// TIA Portal V20 export
// export: Created 2025-12-01T14:57:41.3483873Z, ExportSetting None, DisplayName Totally Integrated Automation Portal, DisplayVersion V20 Update 3, DisplayName TIA Portal Openness, DisplayVersion V20 Update 3, DisplayName TIA Portal Version Control Interface, DisplayVersion V20 Update 3, DisplayName STEP 7 Professional, DisplayVersion V20 Update 3, DisplayName STEP 7 Safety, DisplayVersion V20 Update 2, DisplayName WinCC Basic/Comfort/Advanced, DisplayVersion V20 Update 3, DisplayName WinCC Professional, DisplayVersion V20 Update 3, DisplayName WinCC Unified, DisplayVersion V20 Update 3
FUNCTION_BLOCK "FB380_PaletizadorLenze_NDD"   // FB380, LAD
{ S7_Optimized_Access := 'FALSE' }
// stored: AutoNumber false, SetENOAutomatically false
   VAR_INPUT
      MesaElevador : UInt;
      MesaHorquilla : UInt;
      MesaGarra : UInt;
      NDB_ConfigNDD : UInt;
      NDB_DatosNDD : UInt;
      NDB_Enfardadora : UInt;
      Error_Tx : Bool;
      DesHabilitar_MAQ : Bool;
      DesHabilitar_Enfadadora : Bool;
      DesHabilitar_Horquilla : Bool;   // DesHabilitar la Horquilla
      DesHabilitar_Garra : Bool;   // DesHabilitar la Garra
      PorCapas_Enfardado : Bool;
      Mantenimiento : Bool;
      TermicoFRENO_Elev : Bool;
      Elev_Protusion : Bool;
      EM_Elev_Down : Bool;
      CheckElev_EnEntrada : Bool;
      CheckElev_EnSalida : Bool;
      CheckElev_EnEnfardadora : Bool;
      CheckElev_EnHorquilla : Bool;
      CheckElev_EnGarra : Bool;
      EM_Elev_Up : Bool;
      EM_Elev_Bulon_Dch : Bool;
      EM_Elev_Bulon_Izq : Bool;
      P_Puesto_Capa : Bool;
      P_Puesto_Subir : Bool;
      P_Puesto_Bajar : Bool;
      BarreraNivelUp : Bool;
      BarreraNivelDown : Bool;
      Elev_Galibo_01 : Bool;
      Elev_Galibo_02 : Bool;
      Elev_Galibo_03 : Bool;
      Elev_Galibo_04 : Bool;
      Manual_ElevUp : Bool;
      Manual_ElevDown : Bool;
      Homming_Elev : Bool;
      ModoEncoder_Elev : Bool;
      pHsRef_Elev : Bool;
      V_TOut_Elevacion : Time;
      V_TMP_Protusion : Time;
   END_VAR
   VAR_OUTPUT
      DI3VarElev_pHsReferenciaCero : Bool;
      DesHabiBarreraNivelUP : Bool;
      DesHabiBarreraNivelDown : Bool;
   END_VAR
   VAR
      FB_Enfardadora { S7_SetPoint := 'True'} : "FB384_Enfardadora_Paletizador_NDD";
      Interlock_Horquilla { S7_SetPoint := 'True'} : "NDD_Interlock_Horquilla";
      Interlock_Garras { S7_SetPoint := 'True'} : "NDD_Interlock_Garras";
      Interlock_TELEV { S7_SetPoint := 'True'} : "NDD_Interlock_TElev";
      Ordenes { S7_SetPoint := 'True'} : "NDD_Ordenes";
      TMPEnPisoCarga { S7_SetPoint := 'True'} : TON_TIME;
      TMPEnPisoDesCarga { S7_SetPoint := 'True'} : TON_TIME;
      TMPEnPisoHorquilla { S7_SetPoint := 'True'} : TON_TIME;
      TMPEnPisoGarra { S7_SetPoint := 'True'} : TON_TIME;
      TMPEnPisoEnfradadora { S7_SetPoint := 'True'} : TON_TIME;
      TEstableMovElev { S7_SetPoint := 'True'} : TON_TIME;
      TMPGalibo { S7_SetPoint := 'True'} : TON_TIME;
      TMPProtusion { S7_SetPoint := 'True'} : TON_TIME;
      TOutElevacion { S7_SetPoint := 'True'} : TON_TIME;
      TEsperaMoverElev { S7_SetPoint := 'True'} : TON_TIME;
      TOutPosicion { S7_SetPoint := 'True'} : TON_TIME;
      VelocidadEnfardadora : Int;
      MemoAlturaPedido : Int;
      MemoEventoPaletizado : UInt;
      AlturaActualPedido : Int;
      PosicionCarga : Int;
      PosicionDesCarga : Int;
      PosicionEnfardado : Int;
      PosicionHorquilla : Int;
      PosicionGarra : Int;
      PosicionActual : Int;
      PosicionMoverElev : Int;
      PosicionUltimaElev : Int;
      ConsignaFR_elev : Int;
      SubjectArea_Elev : Word;
      IDArea_Elev : Word;
      MoverElev : Bool;
      FinMoverElev : Bool;
      MFinMoverElev : Bool;
      PosCarga_OK : Bool;
      PosDesCarga_OK : Bool;
      PosHorquilla_OK : Bool;
      PosGarra_OK : Bool;
      PosEnfardadora_OK : Bool;
      TestAuto_HorqGarra : Bool;
      ELEV_ET00 : Bool;
      ELEV_ET01 : Bool;
      CARGA_ET01 : Bool;
      CARGA_ET02 : Bool;
      CARGA_ET03 : Bool;
      CARGA_ET04 : Bool;
      CARGARRA_ET01 : Bool;
      CARGARRA_ET02 : Bool;
      CARGARRA_ET03 : Bool;
      CARGARRA_ET04 : Bool;
      CARGARRA_ET05 : Bool;
      DCARGARRA_ET01 : Bool;
      DCARGARRA_ET02 : Bool;
      DCARGARRA_ET03 : Bool;
      DCARGARRA_ET04 : Bool;
      DCARGARRA_ET05 : Bool;
      DCARHORQ_ET01 : Bool;
      DCARHORQ_ET02 : Bool;
      DCARHORQ_ET03 : Bool;
      DCARHORQ_ET04 : Bool;
      DCARHORQ_ET05 : Bool;
      PALETIZAR_ET01 : Bool;
      PALETIZAR_ET02 : Bool;
      PALETIZAR_ER01 : Bool;
      PALETIZAR_ER02 : Bool;
      DESCARGA_ET02 : Bool;
      DESCARGA_ET03 : Bool;
      DESCARGA_ET04 : Bool;
      DESCARGA_ET05 : Bool;
      DESCARGA_ET06 : Bool;
      MoverElev_Entrada : Bool;
      MoverElev_Garra : Bool;
      MoverElev_HorquillaUp : Bool;
      MoverElev_HorquillaDown : Bool;
      MoverElev_Enfardado : Bool;
      MoverElev_Salida : Bool;
      MoverElev_Puesto : Bool;
      HorqGarra_EnOperacion : Bool;
      Elev_EnReset : Bool;
      Elev_EnReposo : Bool;
      Elev_CargaDeEntrada : Bool;
      Elev_CargaDeGarra : Bool;
      Elev_DesCargaEnGarra : Bool;
      Elev_DesCargaEnHorquilla : Bool;
      Elev_DesCargaEnSalida : Bool;
      Elev_Paletizando : Bool;
      PuestoCarga_EnElev : Bool;
      Memo_NuevaCapa : Bool;
      MA_Puesto_NuevaCapa : Bool;
      MA_Puesto_Subir : Bool;
      MA_Puesto_Bajar : Bool;
      MA_Puesto_Baliza : Bool;
      LibreZonaAlta : Bool;
      ErrorVariador_Elev : Bool;
      MemoHoming_Elev : Bool;
      ReferenciaOK_Elev : Bool;
      MovHorq_Bloqueada : Bool;
      MovGarra_Bloqueada : Bool;
      ErrorControlPedido : Bool;
      AvisoControlPedido : Bool;
      EventoInicioPaletizado : Bool;
      EventoFinalPaletizado : Bool;
      EventoAlturaPedido : Bool;
      EventoInicioEnfardado : Bool;
      EventoFinalEnfardado : Bool;
      EventoErrorEnfradado : Bool;
   END_VAR
   VAR_TEMP
      EstadoZonaMaquina : "EstadoZona";
      EstadoZonaMesa : "EstadoZona";
      EstadoVI : "EstadosMesa_Transporte_Paletizador_NDD";
      EstadoMAQ : "EstadoMaquina_PaletizadorLenze_NDD";
      EstadoHorquilla : "EstadosMesa_HorquillaLenze_Paletizador_NDD";
      EstadoGarra : "EstadosMesa_GarrasLenze_Paletizador_NDD";
      DatosEscada : "UDT_ScadaDatosMaquina";
      EstadoZonaEnfa : "EstadoZona";
      EstadoZonaMovElev : "EstadoZona";
      NodoVar_Elev : "Status_NodosProfinet";
      P_EstadoZonaEnfa : DWord;
      P_EstadoZonaMovElev : DWord;
      P_NodoVar_Elev : DWord;
      Guardar_AR1 : DWord;
      Guardar_AR2 : DWord;
      P_Temporal : DWord;
      DB_ConfigNDD : Word;
      DB_DatosNDD : Word;
      NumDB_DiagProfinet : UInt;
      NumDB_DatosDanfoss : UInt;
      ByteInicial_VarElev : UInt;
      NumNodo_VarElev : UInt;
      VeloManual : Int;   // Velocidad Manual
      VeloCapa : Int;   // Velocidad Nueva Capa
      VeloRapidaDOWN : Int;   // Velocidad Rapida para ir a Posicion DOWN
      VeloLentaDOWN : Int;   // Velocidad Lenta para ir a Posicion DOWN
      PosLentaDOWN : Int;   // Diferencia para pasar Lenta para ir a Posicion DOWN
      VeloRapidaUP : Int;   // Velocidad Rapida para ir a Posicion UP
      VeloLentaUP : Int;   // Velocidad Lenta para ir a Posicion UP
      PosLentaUP : Int;   // Diferencia para pasar Lenta para ir a Posicion UP
      FactorVelocidadEnfardadora : Int;
      AltNivelCtr : Int;
      AlturaMax : Int;
      AlturaMin : Int;
      AlturaPaleta : Int;
      AlturaGalibo : Int;
      AlturaMaximoPedido : Int;
      AlturaControlPedido : Int;
      PosicionLibreNDD : Int;
      PosicionLibreHorq : Int;
      PosicionLibreGarra : Int;
      MemoPosActual_Elev : Int;
      MargenPos : Int;
      AuxPosMax : Int;
      AuxPosMin : Int;
      MargenPedido : Int;
      AuxAlturaPedidoMax : Int;
      AuxAlturaPedidoMin : Int;
      TempInt : Int;
      OrdenPosUP : Bool;
      OrdenPosDOWN : Bool;
      OrdenPosLentaUP : Bool;
      OrdenPosLentaDown : Bool;
      ZonaEnMarcha : Bool;
      ZonaEnReset : Bool;
      ZonaEnParoBlando : Bool;
      EnPisoAbajo : Bool;
      NodoNoPres_VarElev : Bool;
      AuxEstados : Bool;
      Etapas_OK : Bool;
      Transicion_OK : Bool;
      ControlPaleta_OK : Bool;
      AlturaMaxOK_Puesto : Bool;
      AlturaMinOK_Puesto : Bool;
      DesHabilitar_NDD : Bool;
      CalcularAlturaPedido : Bool;
   END_VAR
   VAR_TEMP   // added for the SCL form of the ladder/FBD networks
      _w1 : Bool;
      _w2 : Bool;
      _w3 : Bool;
      _w4 : Bool;
      _w5 : Bool;
      _w6 : Bool;
      _w7 : Bool;
   END_VAR
BEGIN

REGION Network 1: Variables de Testeo en Automatico
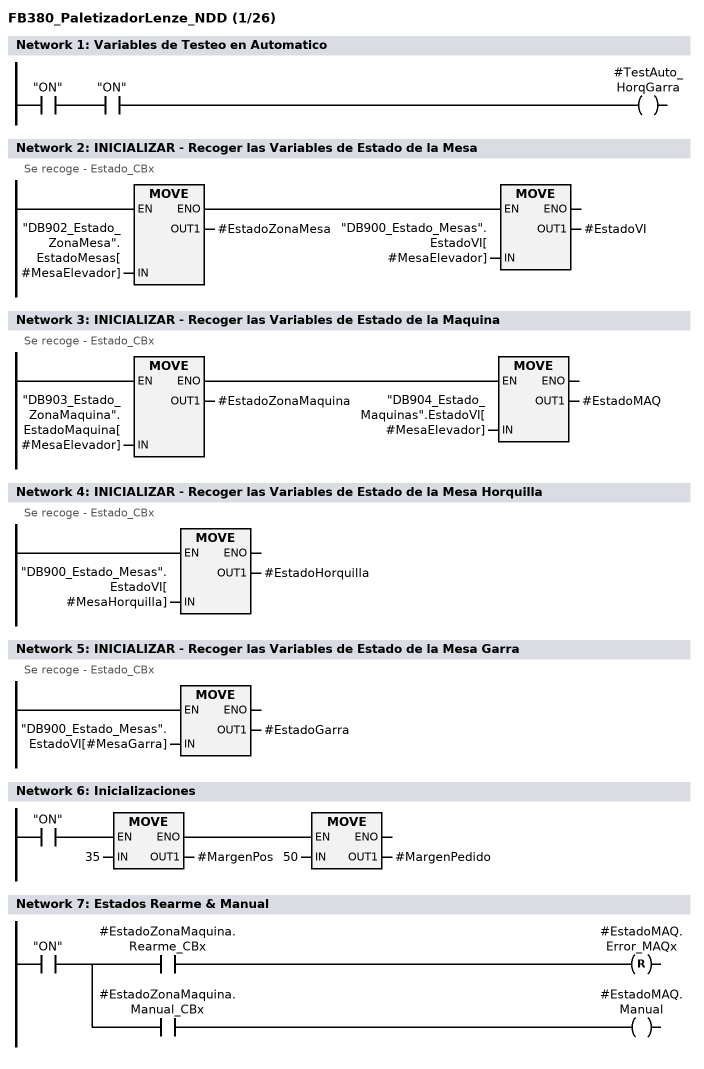
   RUNG wire#powerrail
      Contact( "ON" )
      Contact( "ON" )
      Coil( #TestAuto_HorqGarra )
   END_RUNG
   // the same network as SCL:
   #TestAuto_HorqGarra := "ON" AND "ON";
END_REGION

REGION Network 2: INICIALIZAR - Recoger las Variables de Estado de la Mesa
   // Se recoge - Estado_CBx
   RUNG wire#powerrail
      Move(in := "DB902_Estado_ZonaMesa".EstadoMesas[#MesaElevador], out1 => #EstadoZonaMesa)
      Move(in := "DB900_Estado_Mesas".EstadoVI[#MesaElevador], out1 => #EstadoVI)
   END_RUNG
   // the same network as SCL:
   #EstadoZonaMesa := "DB902_Estado_ZonaMesa".EstadoMesas[#MesaElevador];
   #EstadoVI := "DB900_Estado_Mesas".EstadoVI[#MesaElevador];
END_REGION

REGION Network 3: INICIALIZAR - Recoger las Variables de Estado de la Maquina
   // Se recoge - Estado_CBx
   RUNG wire#powerrail
      Move(in := "DB903_Estado_ZonaMaquina".EstadoMaquina[#MesaElevador], out1 => #EstadoZonaMaquina)
      Move(in := "DB904_Estado_Maquinas".EstadoVI[#MesaElevador], out1 => #EstadoMAQ)
   END_RUNG
   // the same network as SCL:
   #EstadoZonaMaquina := "DB903_Estado_ZonaMaquina".EstadoMaquina[#MesaElevador];
   #EstadoMAQ := "DB904_Estado_Maquinas".EstadoVI[#MesaElevador];
END_REGION

REGION Network 4: INICIALIZAR - Recoger las Variables de Estado de la Mesa Horquilla
   // Se recoge - Estado_CBx
   RUNG wire#powerrail
      Move(in := "DB900_Estado_Mesas".EstadoVI[#MesaHorquilla], out1 => #EstadoHorquilla)
   END_RUNG
   // the same network as SCL:
   #EstadoHorquilla := "DB900_Estado_Mesas".EstadoVI[#MesaHorquilla];
END_REGION

REGION Network 5: INICIALIZAR - Recoger las Variables de Estado de la Mesa Garra
   // Se recoge - Estado_CBx
   RUNG wire#powerrail
      Move(in := "DB900_Estado_Mesas".EstadoVI[#MesaGarra], out1 => #EstadoGarra)
   END_RUNG
   // the same network as SCL:
   #EstadoGarra := "DB900_Estado_Mesas".EstadoVI[#MesaGarra];
END_REGION

REGION Network 6: Inicializaciones
   RUNG wire#powerrail
      Contact( "ON" )
      { S7_GenerateENO := "TRUE" } Move(in := 35, out1 => #MargenPos)
      { S7_GenerateENO := "TRUE" } Move(in := 50, out1 => #MargenPedido)
   END_RUNG
   // the same network as SCL:
   // ENO of a box is taken as its EN; it also drops when the box reports an error
   IF "ON" THEN
       #MargenPos := 35;
       #MargenPedido := 50;
   END_IF;
END_REGION

REGION Network 7: Estados Rearme & Manual
   RUNG wire#powerrail
      Contact( "ON" )
      wire#w1
      Contact( #EstadoZonaMaquina.Rearme_CBx )
      R_Coil( #EstadoMAQ.Error_MAQx )
   END_RUNG
   RUNG wire#w1
      Contact( #EstadoZonaMaquina.Manual_CBx )
      Coil( #EstadoMAQ.Manual )
   END_RUNG
   // the same network as SCL:
   IF "ON" AND #EstadoZonaMaquina.Rearme_CBx THEN #EstadoMAQ.Error_MAQx := FALSE; END_IF;
   #EstadoMAQ.Manual := "ON" AND #EstadoZonaMaquina.Manual_CBx;
END_REGION

REGION Network 8: Deshabilitar NDD
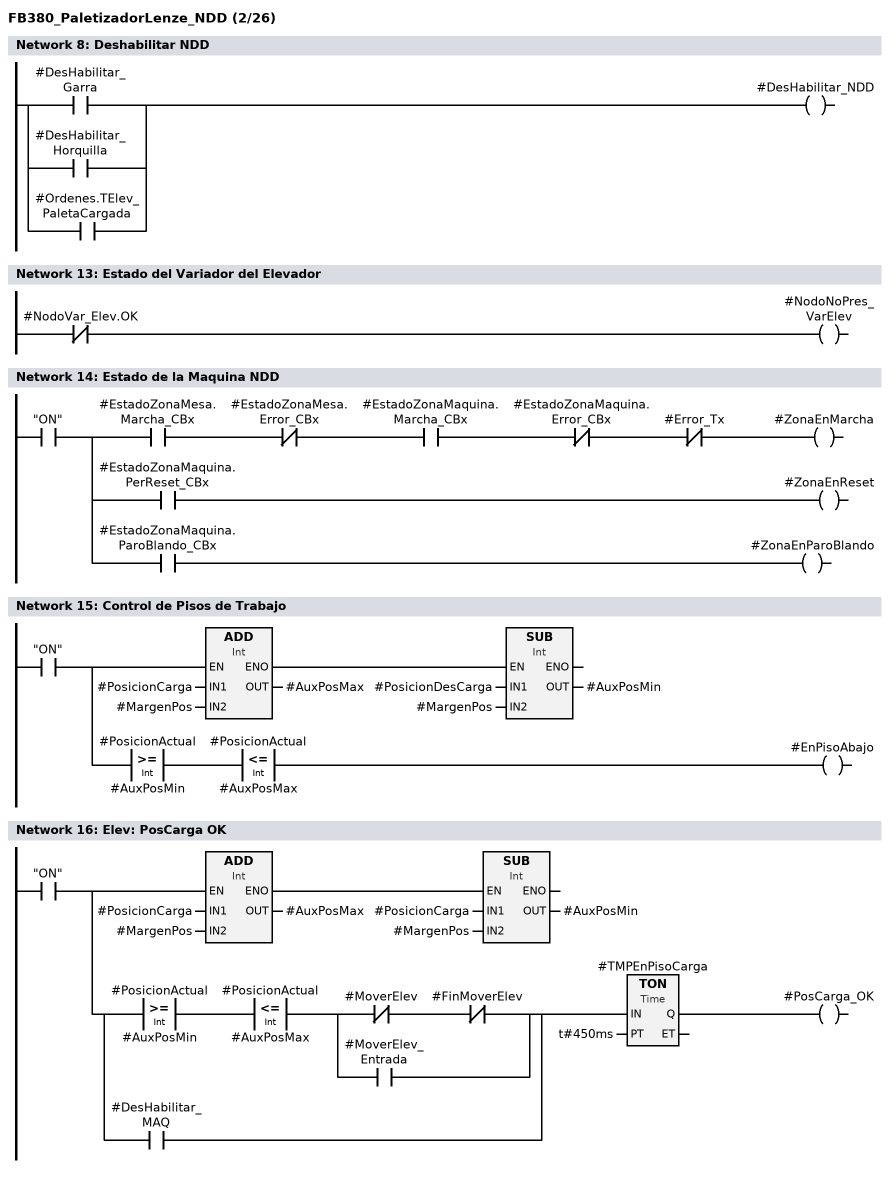
   RUNG wire#powerrail
      Contact( #DesHabilitar_Garra )
      wire#w1
      Coil( #DesHabilitar_NDD )
   END_RUNG
   RUNG wire#powerrail
      Contact( #DesHabilitar_Horquilla )
   END_RUNG wire#w1
   RUNG wire#powerrail
      Contact( #Ordenes.TElev_PaletaCargada )
   END_RUNG wire#w1
   // the same network as SCL:
   #DesHabilitar_NDD := #DesHabilitar_Garra OR #DesHabilitar_Horquilla OR #Ordenes.TElev_PaletaCargada;
END_REGION

NETWORK
TITLE = Datos Internos del Elevador
/////////////////////////////////////////////////////////////////////////////
/////////////////////////////////////////////////////////////////////////////
// - Inicializaciones Previas

      TAR1  #Guardar_AR1;  // - Guardar el AR1


/////////////////////////////////////////////////////////////////////////////
/////////////////////////////////////////////////////////////////////////////
// - Recoger datos Previos del Elevador

      L     #NDB_ConfigNDD;  // - DB's de configuracion del Elevador
      T     #DB_ConfigNDD;  //   DB General
      L     #NDB_DatosNDD;  //   DB Particular
      T     #DB_DatosNDD;


/////////////////////////////////////////////////////////////////////////////
/////////////////////////////////////////////////////////////////////////////
// --- Sistema de Profinet

      LAR1  P#0.0;  // - Leer Datos de los Variadores
      OPN   DB [#DB_DatosNDD];  //   del NDD

      L     DBW [AR1, P#0.0];  // - Num DB de Profinet
      T     #NumDB_DiagProfinet;
      L     DBW [AR1, P#2.0];  // - Num DB de DANFOSS
      T     #NumDB_DatosDanfoss;

      L     DBW [AR1, P#4.0];  // - Nodos de los Variadores
      T     #NumNodo_VarElev;


      L     DBW [AR1, P#10.0];  // - Direcciones de los Variadores
      T     #ByteInicial_VarElev;

      L     P##NodoVar_Elev;  // Puntero del Estado del Nodo del Variador de Elevador (TEMPORAL)
      T     #P_NodoVar_Elev;



NETWORK
TITLE = --- Velocidades y Posiciones
/////////////////////////////////////////////////////////////////////////////
/////////////////////////////////////////////////////////////////////////////
// - Recoger Datos Generales del Elevador

      LAR1  P#0.0;  // - Leer Datos de Velocidad
      OPN   DB [#DB_ConfigNDD];

      L     DBW [AR1, P#0.0];  //   Velocidad Manual
      T     #VeloManual;
      L     DBW [AR1, P#2.0];  //   Velocidad Capa
      T     #VeloCapa;

      L     DBW [AR1, P#4.0];  //   Velocidades del Movimiento hacia DOWN
      T     #VeloRapidaDOWN;
      L     DBW [AR1, P#6.0];
      T     #VeloLentaDOWN;

      L     DBW [AR1, P#8.0];  //   Velocidades del Movimiento hacia UP
      T     #VeloRapidaUP;
      L     DBW [AR1, P#10.0];
      T     #VeloLentaUP;

      L     DBW [AR1, P#12.0];  //   Posiciones de Cambio de velocidad
      T     #PosLentaDOWN;
      L     DBW [AR1, P#14.0];
      T     #PosLentaUP;


/////////////////////////////////////////////////////////////////////////////
/////////////////////////////////////////////////////////////////////////////
// - Recoger Datos Particulares de cada Elevador

      LAR1  P#16.0;  // - Leer Datos de de funcionamiento
      OPN   DB [#DB_DatosNDD];  //   del Elevador

      L     DBW [AR1, P#0.0];  // - Configuracion Fisica
      T     #AlturaMax;
      L     DBW [AR1, P#2.0];
      T     #AlturaMin;
      L     DBW [AR1, P#4.0];
      T     #AlturaPaleta;
      L     DBW [AR1, P#6.0];
      T     #AlturaGalibo;

      L     DBW [AR1, P#8.0];  // - Posiciones de Transferencia
      T     #PosicionCarga;
      L     DBW [AR1, P#10.0];
      T     #PosicionDesCarga;
      L     DBW [AR1, P#12.0];
//      L     #FB_Enfardadora.PosicionEnfardado
      T     #PosicionEnfardado;
      L     DBW [AR1, P#14.0];
      T     #PosicionHorquilla;
      L     DBW [AR1, P#16.0];
      T     #PosicionGarra;

      L     DBW [AR1, P#18.0];  // - Configuracion de Liberación del Elevador
      T     #PosicionLibreNDD;
      L     DBW [AR1, P#20.0];
      T     #PosicionLibreHorq;
      L     DBW [AR1, P#22.0];
      T     #PosicionLibreGarra;


      L     DBW [AR1, P#24.0];  // - Configuracion del Pedido
      T     #AlturaMaximoPedido;
      L     DBW [AR1, P#26.0];
      T     #AlturaControlPedido;

      L     DBW [AR1, P#28.0];  // - Factor de la Velocidad enviado por la Enfardadora
      T     #FactorVelocidadEnfardadora;

      L     #AlturaMax;  // - Altura para DesActivar el control de la Barrera
      L     200;
      -I;
      T     #AltNivelCtr;




NETWORK
TITLE = --- Nodo PROFINET >>> Estado
// ------------------------------------------------------------------------------------
// ------------------------------------------------------------------------------------
// --- Estado del Nodo de PROFINET del Variador de la Elevador (LENZE)

      L     #NumNodo_VarElev;  // Nodo de Profinet
      L     1;
      -I;
      L     2;  // Longitud registro datos
      *I;
      SLD   3;
      LAR1;

      OPN   DB [#NumDB_DiagProfinet];  // Leer estado del Nodo de PROFINET
      L     DBW [AR1, P#0.0];
      T     LW [#P_NodoVar_Elev];



NETWORK
TITLE = ---
/////////////////////////////////////////////////////////////////////////////
/////////////////////////////////////////////////////////////////////////////
// - Final de la Recogida de Datos del Elevador

      LAR1  #Guardar_AR1;  // - Recuperar AR1



REGION Network 13: Estado del Variador del Elevador
   RUNG wire#powerrail
      I_Contact( #NodoVar_Elev.OK )
      Coil( #NodoNoPres_VarElev )
   END_RUNG
   // the same network as SCL:
   #NodoNoPres_VarElev := NOT #NodoVar_Elev.OK;
END_REGION

REGION Network 14: Estado de la Maquina NDD
   RUNG wire#powerrail
      Contact( "ON" )
      wire#w1
      Contact( #EstadoZonaMesa.Marcha_CBx )
      I_Contact( #EstadoZonaMesa.Error_CBx )
      Contact( #EstadoZonaMaquina.Marcha_CBx )
      I_Contact( #EstadoZonaMaquina.Error_CBx )
      I_Contact( #Error_Tx )
      Coil( #ZonaEnMarcha )
   END_RUNG
   RUNG wire#w1
      Contact( #EstadoZonaMaquina.PerReset_CBx )
      Coil( #ZonaEnReset )
   END_RUNG
   RUNG wire#w1
      Contact( #EstadoZonaMaquina.ParoBlando_CBx )
      Coil( #ZonaEnParoBlando )
   END_RUNG
   // the same network as SCL:
   #ZonaEnMarcha := "ON" AND #EstadoZonaMesa.Marcha_CBx AND NOT #EstadoZonaMesa.Error_CBx AND #EstadoZonaMaquina.Marcha_CBx AND NOT #EstadoZonaMaquina.Error_CBx AND NOT #Error_Tx;
   #ZonaEnReset := "ON" AND #EstadoZonaMaquina.PerReset_CBx;
   #ZonaEnParoBlando := "ON" AND #EstadoZonaMaquina.ParoBlando_CBx;
END_REGION

REGION Network 15: Control de Pisos de Trabajo
   RUNG wire#powerrail
      Contact( "ON" )
      wire#w1
      { S7_Templates := "SrcType := Int"; S7_GenerateENO := "TRUE" } Add(in1 := #PosicionCarga, in2 := #MargenPos, out => #AuxPosMax)
      { S7_Templates := "SrcType := Int"; S7_GenerateENO := "TRUE" } Sub(in1 := #PosicionDesCarga, in2 := #MargenPos, out => #AuxPosMin)
   END_RUNG
   RUNG wire#w1
      { S7_Templates := "SrcType := Int" } GE_Contact(in1 := #PosicionActual, in2 := #AuxPosMin)
      { S7_Templates := "SrcType := Int" } LE_Contact(in1 := #PosicionActual, in2 := #AuxPosMax)
      Coil( #EnPisoAbajo )
   END_RUNG
   // the same network as SCL:
   // ENO of a box is taken as its EN; it also drops when the box reports an error
   IF "ON" THEN
       #AuxPosMax := #PosicionCarga + #MargenPos;
       #AuxPosMin := #PosicionDesCarga - #MargenPos;
   END_IF;
   #EnPisoAbajo := "ON" AND (#PosicionActual >= #AuxPosMin) AND (#PosicionActual <= #AuxPosMax);
END_REGION

REGION Network 16: Elev: PosCarga OK
   RUNG wire#powerrail
      Contact( "ON" )
      wire#w1
      { S7_Templates := "SrcType := Int"; S7_GenerateENO := "TRUE" } Add(in1 := #PosicionCarga, in2 := #MargenPos, out => #AuxPosMax)
      { S7_Templates := "SrcType := Int"; S7_GenerateENO := "TRUE" } Sub(in1 := #PosicionCarga, in2 := #MargenPos, out => #AuxPosMin)
   END_RUNG
   RUNG wire#w1
      { S7_Templates := "SrcType := Int" } GE_Contact(in1 := #PosicionActual, in2 := #AuxPosMin)
      { S7_Templates := "SrcType := Int" } LE_Contact(in1 := #PosicionActual, in2 := #AuxPosMax)
      wire#w2
      I_Contact( #MoverElev )
      I_Contact( #FinMoverElev )
      wire#w3
      { S7_Templates := "time_type := Time" } #TMPEnPisoCarga.TON(pt := t#450ms, et =>)
      Coil( #PosCarga_OK )
   END_RUNG
   RUNG wire#w2
      Contact( #MoverElev_Entrada )
   END_RUNG wire#w3
   RUNG wire#w1
      Contact( #DesHabilitar_MAQ )
   END_RUNG wire#w3
   // the same network as SCL:
   // ENO of a box is taken as its EN; it also drops when the box reports an error
   IF "ON" THEN
       #AuxPosMax := #PosicionCarga + #MargenPos;
       #AuxPosMin := #PosicionCarga - #MargenPos;
   END_IF;
   #TMPEnPisoCarga(IN := "ON" AND (((#PosicionActual >= #AuxPosMin) AND (#PosicionActual <= #AuxPosMax) AND ((NOT #MoverElev AND NOT #FinMoverElev) OR #MoverElev_Entrada)) OR #DesHabilitar_MAQ),   // TON
                   PT := t#450ms);
   #PosCarga_OK := #TMPEnPisoCarga.Q;
END_REGION

REGION Network 17: Elev: PosDesCarga OK
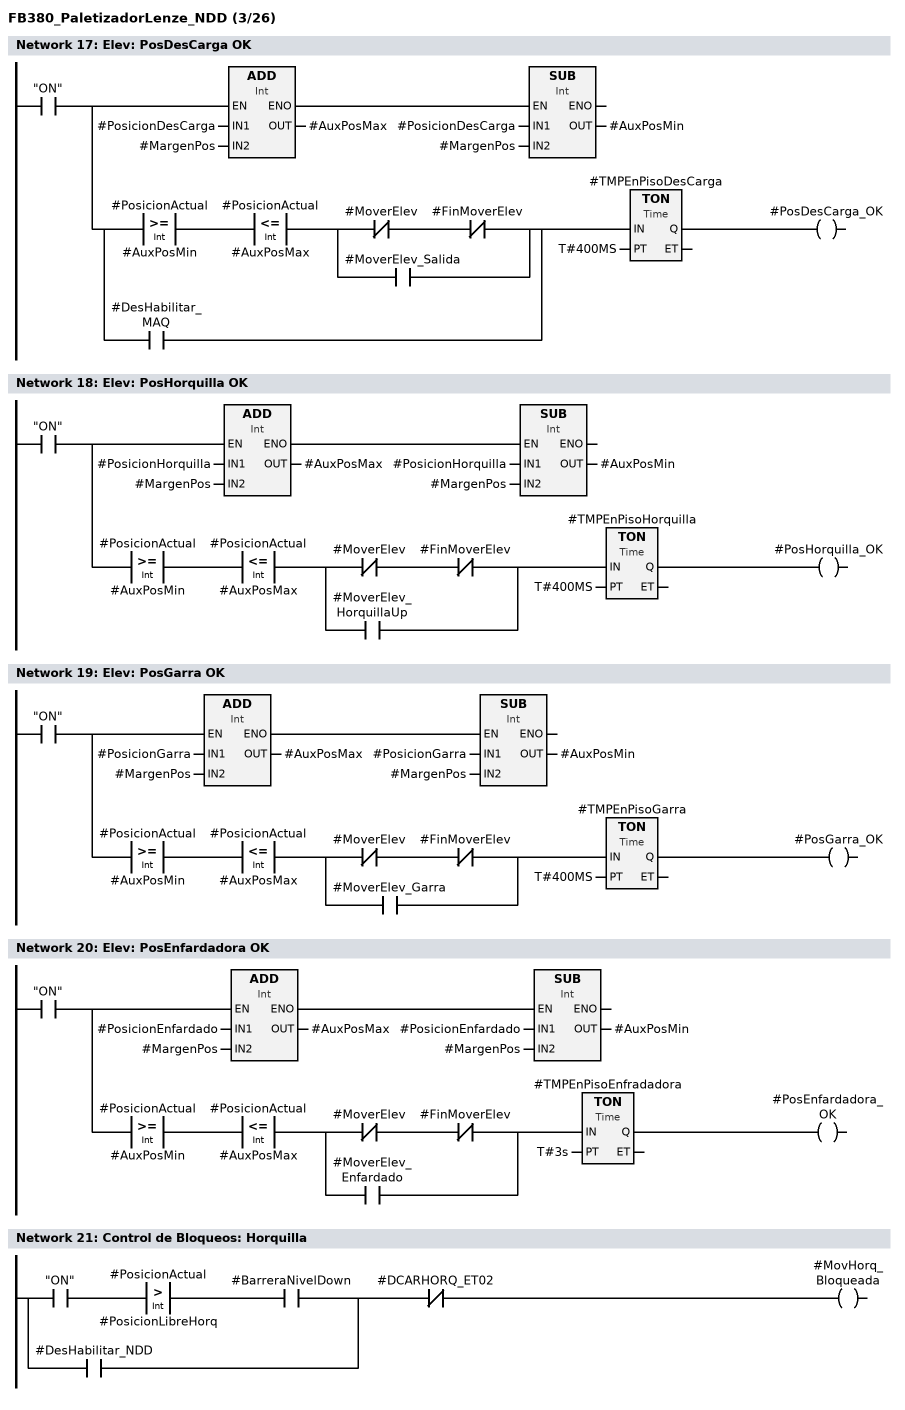
   RUNG wire#powerrail
      Contact( "ON" )
      wire#w1
      { S7_Templates := "SrcType := Int"; S7_GenerateENO := "TRUE" } Add(in1 := #PosicionDesCarga, in2 := #MargenPos, out => #AuxPosMax)
      { S7_Templates := "SrcType := Int"; S7_GenerateENO := "TRUE" } Sub(in1 := #PosicionDesCarga, in2 := #MargenPos, out => #AuxPosMin)
   END_RUNG
   RUNG wire#w1
      { S7_Templates := "SrcType := Int" } GE_Contact(in1 := #PosicionActual, in2 := #AuxPosMin)
      { S7_Templates := "SrcType := Int" } LE_Contact(in1 := #PosicionActual, in2 := #AuxPosMax)
      wire#w2
      I_Contact( #MoverElev )
      I_Contact( #FinMoverElev )
      wire#w3
      { S7_Templates := "time_type := Time" } #TMPEnPisoDesCarga.TON(pt := T#400MS, et =>)
      Coil( #PosDesCarga_OK )
   END_RUNG
   RUNG wire#w2
      Contact( #MoverElev_Salida )
   END_RUNG wire#w3
   RUNG wire#w1
      Contact( #DesHabilitar_MAQ )
   END_RUNG wire#w3
   // the same network as SCL:
   // ENO of a box is taken as its EN; it also drops when the box reports an error
   IF "ON" THEN
       #AuxPosMax := #PosicionDesCarga + #MargenPos;
       #AuxPosMin := #PosicionDesCarga - #MargenPos;
   END_IF;
   #TMPEnPisoDesCarga(IN := "ON" AND (((#PosicionActual >= #AuxPosMin) AND (#PosicionActual <= #AuxPosMax) AND ((NOT #MoverElev AND NOT #FinMoverElev) OR #MoverElev_Salida)) OR #DesHabilitar_MAQ),   // TON
                      PT := T#400MS);
   #PosDesCarga_OK := #TMPEnPisoDesCarga.Q;
END_REGION

REGION Network 18: Elev: PosHorquilla OK
   RUNG wire#powerrail
      Contact( "ON" )
      wire#w1
      { S7_Templates := "SrcType := Int"; S7_GenerateENO := "TRUE" } Add(in1 := #PosicionHorquilla, in2 := #MargenPos, out => #AuxPosMax)
      { S7_Templates := "SrcType := Int"; S7_GenerateENO := "TRUE" } Sub(in1 := #PosicionHorquilla, in2 := #MargenPos, out => #AuxPosMin)
   END_RUNG
   RUNG wire#w1
      { S7_Templates := "SrcType := Int" } GE_Contact(in1 := #PosicionActual, in2 := #AuxPosMin)
      { S7_Templates := "SrcType := Int" } LE_Contact(in1 := #PosicionActual, in2 := #AuxPosMax)
      wire#w2
      I_Contact( #MoverElev )
      I_Contact( #FinMoverElev )
      wire#w3
      { S7_Templates := "time_type := Time" } #TMPEnPisoHorquilla.TON(pt := T#400MS, et =>)
      Coil( #PosHorquilla_OK )
   END_RUNG
   RUNG wire#w2
      Contact( #MoverElev_HorquillaUp )
   END_RUNG wire#w3
   // the same network as SCL:
   // ENO of a box is taken as its EN; it also drops when the box reports an error
   IF "ON" THEN
       #AuxPosMax := #PosicionHorquilla + #MargenPos;
       #AuxPosMin := #PosicionHorquilla - #MargenPos;
   END_IF;
   #TMPEnPisoHorquilla(IN := "ON" AND (#PosicionActual >= #AuxPosMin) AND (#PosicionActual <= #AuxPosMax) AND ((NOT #MoverElev AND NOT #FinMoverElev) OR #MoverElev_HorquillaUp),   // TON
                       PT := T#400MS);
   #PosHorquilla_OK := #TMPEnPisoHorquilla.Q;
END_REGION

REGION Network 19: Elev: PosGarra OK
   RUNG wire#powerrail
      Contact( "ON" )
      wire#w1
      { S7_Templates := "SrcType := Int"; S7_GenerateENO := "TRUE" } Add(in1 := #PosicionGarra, in2 := #MargenPos, out => #AuxPosMax)
      { S7_Templates := "SrcType := Int"; S7_GenerateENO := "TRUE" } Sub(in1 := #PosicionGarra, in2 := #MargenPos, out => #AuxPosMin)
   END_RUNG
   RUNG wire#w1
      { S7_Templates := "SrcType := Int" } GE_Contact(in1 := #PosicionActual, in2 := #AuxPosMin)
      { S7_Templates := "SrcType := Int" } LE_Contact(in1 := #PosicionActual, in2 := #AuxPosMax)
      wire#w2
      I_Contact( #MoverElev )
      I_Contact( #FinMoverElev )
      wire#w3
      { S7_Templates := "time_type := Time" } #TMPEnPisoGarra.TON(pt := T#400MS, et =>)
      Coil( #PosGarra_OK )
   END_RUNG
   RUNG wire#w2
      Contact( #MoverElev_Garra )
   END_RUNG wire#w3
   // the same network as SCL:
   // ENO of a box is taken as its EN; it also drops when the box reports an error
   IF "ON" THEN
       #AuxPosMax := #PosicionGarra + #MargenPos;
       #AuxPosMin := #PosicionGarra - #MargenPos;
   END_IF;
   #TMPEnPisoGarra(IN := "ON" AND (#PosicionActual >= #AuxPosMin) AND (#PosicionActual <= #AuxPosMax) AND ((NOT #MoverElev AND NOT #FinMoverElev) OR #MoverElev_Garra),   // TON
                   PT := T#400MS);
   #PosGarra_OK := #TMPEnPisoGarra.Q;
END_REGION

REGION Network 20: Elev: PosEnfardadora OK
   RUNG wire#powerrail
      Contact( "ON" )
      wire#w1
      { S7_Templates := "SrcType := Int"; S7_GenerateENO := "TRUE" } Add(in1 := #PosicionEnfardado, in2 := #MargenPos, out => #AuxPosMax)
      { S7_Templates := "SrcType := Int"; S7_GenerateENO := "TRUE" } Sub(in1 := #PosicionEnfardado, in2 := #MargenPos, out => #AuxPosMin)
   END_RUNG
   RUNG wire#w1
      { S7_Templates := "SrcType := Int" } GE_Contact(in1 := #PosicionActual, in2 := #AuxPosMin)
      { S7_Templates := "SrcType := Int" } LE_Contact(in1 := #PosicionActual, in2 := #AuxPosMax)
      wire#w2
      I_Contact( #MoverElev )
      I_Contact( #FinMoverElev )
      wire#w3
      { S7_Templates := "time_type := Time" } #TMPEnPisoEnfradadora.TON(pt := T#3s, et =>)
      Coil( #PosEnfardadora_OK )
   END_RUNG
   RUNG wire#w2
      Contact( #MoverElev_Enfardado )
   END_RUNG wire#w3
   // the same network as SCL:
   // ENO of a box is taken as its EN; it also drops when the box reports an error
   IF "ON" THEN
       #AuxPosMax := #PosicionEnfardado + #MargenPos;
       #AuxPosMin := #PosicionEnfardado - #MargenPos;
   END_IF;
   #TMPEnPisoEnfradadora(IN := "ON" AND (#PosicionActual >= #AuxPosMin) AND (#PosicionActual <= #AuxPosMax) AND ((NOT #MoverElev AND NOT #FinMoverElev) OR #MoverElev_Enfardado),   // TON
                         PT := T#3s);
   #PosEnfardadora_OK := #TMPEnPisoEnfradadora.Q;
END_REGION

REGION Network 21: Control de Bloqueos: Horquilla
   RUNG wire#powerrail
      Contact( "ON" )
      { S7_Templates := "SrcType := Int" } GT_Contact(in1 := #PosicionActual, in2 := #PosicionLibreHorq)
      Contact( #BarreraNivelDown )
      wire#w1
      I_Contact( #DCARHORQ_ET02 )
      Coil( #MovHorq_Bloqueada )
   END_RUNG
   RUNG wire#powerrail
      Contact( #DesHabilitar_NDD )
   END_RUNG wire#w1
   // the same network as SCL:
   #MovHorq_Bloqueada := (("ON" AND (#PosicionActual > #PosicionLibreHorq) AND #BarreraNivelDown) OR #DesHabilitar_NDD) AND NOT #DCARHORQ_ET02;
END_REGION

REGION Network 22: Control de Bloqueos: Garra
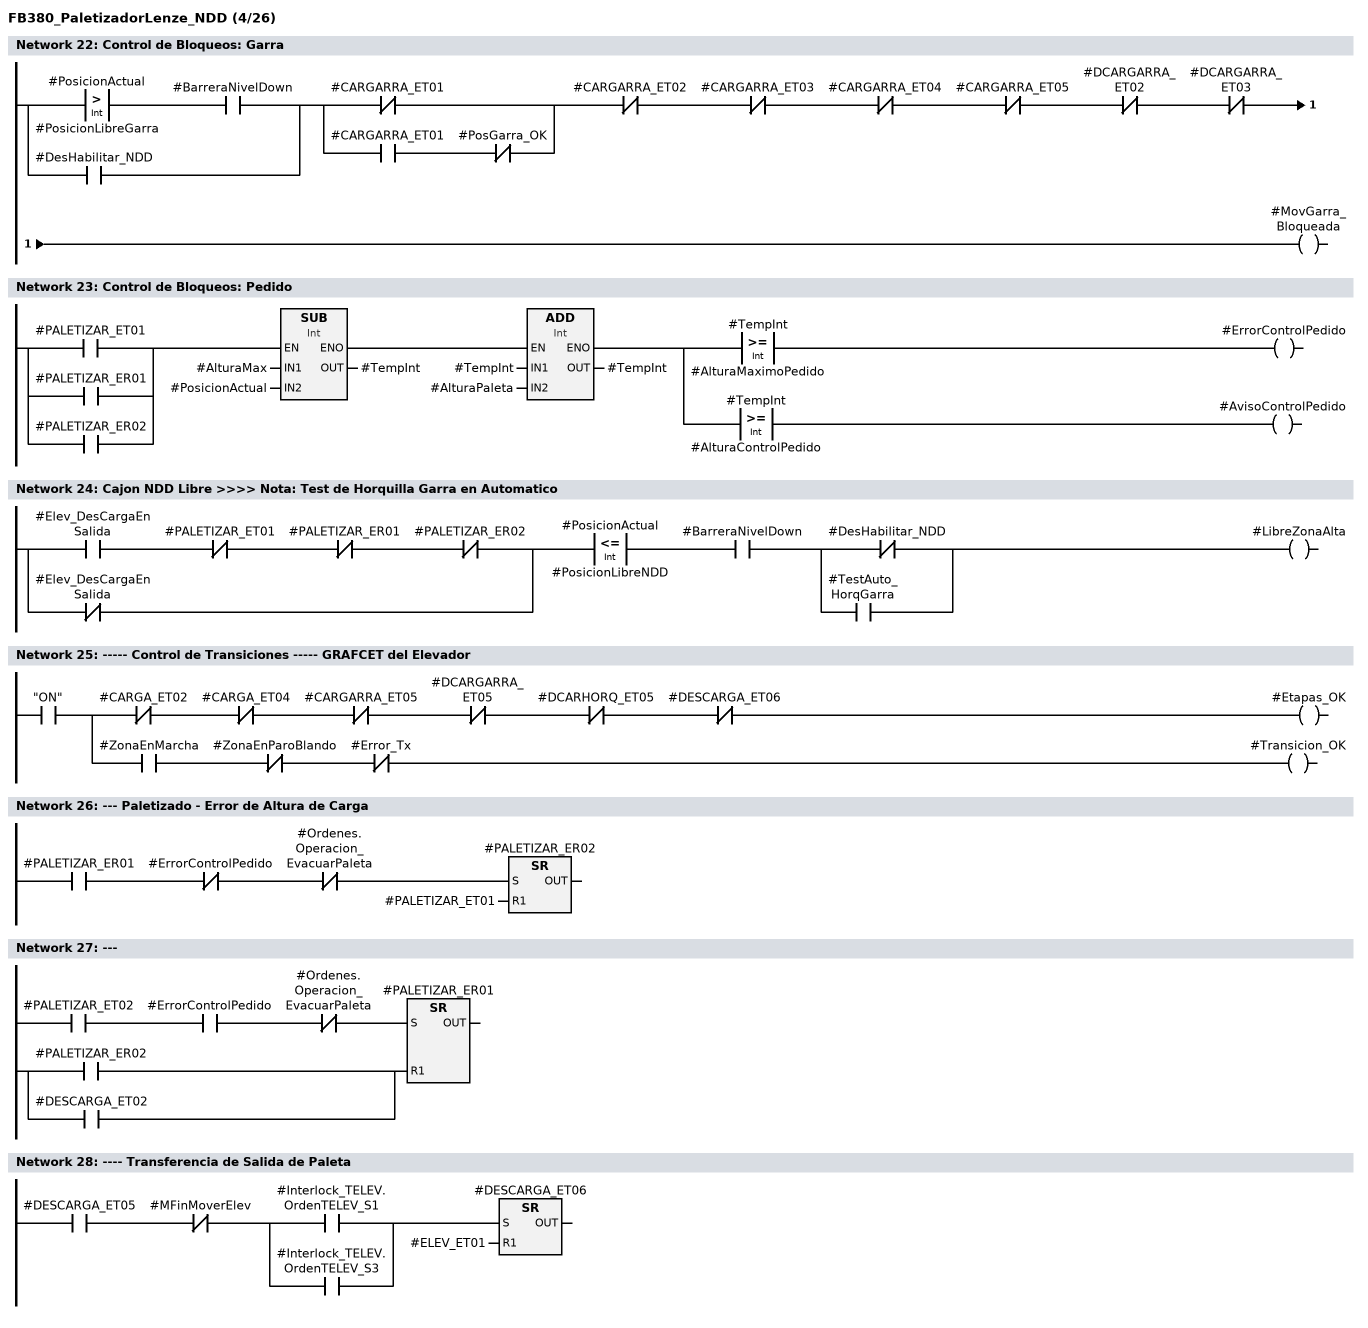
   RUNG wire#powerrail
      { S7_Templates := "SrcType := Int" } GT_Contact(in1 := #PosicionActual, in2 := #PosicionLibreGarra)
      Contact( #BarreraNivelDown )
      wire#w1
      I_Contact( #CARGARRA_ET01 )
      wire#w2
      I_Contact( #CARGARRA_ET02 )
      I_Contact( #CARGARRA_ET03 )
      I_Contact( #CARGARRA_ET04 )
      I_Contact( #CARGARRA_ET05 )
      I_Contact( #DCARGARRA_ET02 )
      I_Contact( #DCARGARRA_ET03 )
      Coil( #MovGarra_Bloqueada )
   END_RUNG
   RUNG wire#powerrail
      Contact( #DesHabilitar_NDD )
   END_RUNG wire#w1
   RUNG wire#w1
      Contact( #CARGARRA_ET01 )
      I_Contact( #PosGarra_OK )
   END_RUNG wire#w2
   // the same network as SCL:
   #MovGarra_Bloqueada := (((#PosicionActual > #PosicionLibreGarra) AND #BarreraNivelDown) OR #DesHabilitar_NDD) AND (NOT #CARGARRA_ET01 OR (#CARGARRA_ET01 AND NOT #PosGarra_OK)) AND NOT #CARGARRA_ET02 AND NOT #CARGARRA_ET03 AND NOT #CARGARRA_ET04 AND NOT #CARGARRA_ET05 AND NOT #DCARGARRA_ET02 AND NOT #DCARGARRA_ET03;
END_REGION

REGION Network 23: Control de Bloqueos: Pedido
   RUNG wire#powerrail
      Contact( #PALETIZAR_ET01 )
      wire#w1
      { S7_Templates := "SrcType := Int"; S7_GenerateENO := "TRUE" } Sub(in1 := #AlturaMax, in2 := #PosicionActual, out => #TempInt)
      { S7_Templates := "SrcType := Int"; S7_GenerateENO := "TRUE" } Add(in1 := #TempInt, in2 := #AlturaPaleta, out => #TempInt)
      wire#w2
      { S7_Templates := "SrcType := Int" } GE_Contact(in1 := #TempInt, in2 := #AlturaMaximoPedido)
      Coil( #ErrorControlPedido )
   END_RUNG
   RUNG wire#powerrail
      Contact( #PALETIZAR_ER01 )
   END_RUNG wire#w1
   RUNG wire#powerrail
      Contact( #PALETIZAR_ER02 )
   END_RUNG wire#w1
   RUNG wire#w2
      { S7_Templates := "SrcType := Int" } GE_Contact(in1 := #TempInt, in2 := #AlturaControlPedido)
      Coil( #AvisoControlPedido )
   END_RUNG
   // the same network as SCL:
   // ENO of a box is taken as its EN; it also drops when the box reports an error
   #_w1 := #PALETIZAR_ET01 OR #PALETIZAR_ER01 OR #PALETIZAR_ER02;
   IF #_w1 THEN
       #TempInt := #AlturaMax - #PosicionActual;
       #TempInt := #TempInt + #AlturaPaleta;
   END_IF;
   #ErrorControlPedido := #_w1 AND (#TempInt >= #AlturaMaximoPedido);
   #AvisoControlPedido := #_w1 AND (#TempInt >= #AlturaControlPedido);
END_REGION

REGION Network 24: Cajon NDD Libre >>>> Nota: Test de Horquilla Garra en Automatico
   RUNG wire#powerrail
      Contact( #Elev_DesCargaEnSalida )
      I_Contact( #PALETIZAR_ET01 )
      I_Contact( #PALETIZAR_ER01 )
      I_Contact( #PALETIZAR_ER02 )
      wire#w1
      { S7_Templates := "SrcType := Int" } LE_Contact(in1 := #PosicionActual, in2 := #PosicionLibreNDD)
      Contact( #BarreraNivelDown )
      wire#w2
      I_Contact( #DesHabilitar_NDD )
      wire#w3
      Coil( #LibreZonaAlta )
   END_RUNG
   RUNG wire#powerrail
      I_Contact( #Elev_DesCargaEnSalida )
   END_RUNG wire#w1
   RUNG wire#w2
      Contact( #TestAuto_HorqGarra )
   END_RUNG wire#w3
   // the same network as SCL:
   #LibreZonaAlta := ((#Elev_DesCargaEnSalida AND NOT #PALETIZAR_ET01 AND NOT #PALETIZAR_ER01 AND NOT #PALETIZAR_ER02) OR NOT #Elev_DesCargaEnSalida) AND (#PosicionActual <= #PosicionLibreNDD) AND #BarreraNivelDown AND (NOT #DesHabilitar_NDD OR #TestAuto_HorqGarra);
END_REGION

REGION Network 25: ----- Control de Transiciones ----- GRAFCET del Elevador
   RUNG wire#powerrail
      Contact( "ON" )
      wire#w1
      I_Contact( #CARGA_ET02 )
      I_Contact( #CARGA_ET04 )
      I_Contact( #CARGARRA_ET05 )
      I_Contact( #DCARGARRA_ET05 )
      I_Contact( #DCARHORQ_ET05 )
      I_Contact( #DESCARGA_ET06 )
      Coil( #Etapas_OK )
   END_RUNG
   RUNG wire#w1
      Contact( #ZonaEnMarcha )
      I_Contact( #ZonaEnParoBlando )
      I_Contact( #Error_Tx )
      Coil( #Transicion_OK )
   END_RUNG
   // the same network as SCL:
   #Etapas_OK := "ON" AND NOT #CARGA_ET02 AND NOT #CARGA_ET04 AND NOT #CARGARRA_ET05 AND NOT #DCARGARRA_ET05 AND NOT #DCARHORQ_ET05 AND NOT #DESCARGA_ET06;
   #Transicion_OK := "ON" AND #ZonaEnMarcha AND NOT #ZonaEnParoBlando AND NOT #Error_Tx;
END_REGION

REGION Network 26: --- Paletizado - Error de Altura de Carga
   RUNG wire#powerrail
      Contact( #PALETIZAR_ER01 )
      I_Contact( #ErrorControlPedido )
      I_Contact( #Ordenes.Operacion_EvacuarPaleta )
      S_SR(operand := #PALETIZAR_ER02, r1 := #PALETIZAR_ET01)
   END_RUNG
   // the same network as SCL:
   IF #PALETIZAR_ER01 AND NOT #ErrorControlPedido AND NOT #Ordenes.Operacion_EvacuarPaleta THEN
       #PALETIZAR_ER02 := TRUE;   // SR flip-flop
   END_IF;
   IF #PALETIZAR_ET01 THEN #PALETIZAR_ER02 := FALSE; END_IF;
END_REGION

REGION Network 27: ---
   RUNG wire#powerrail
      Contact( #PALETIZAR_ET02 )
      Contact( #ErrorControlPedido )
      I_Contact( #Ordenes.Operacion_EvacuarPaleta )
      S_SR(operand := #PALETIZAR_ER01, r1 := wire#w1)
   END_RUNG
   RUNG wire#powerrail
      Contact( #PALETIZAR_ER02 )
   END_RUNG wire#w1
   RUNG wire#powerrail
      Contact( #DESCARGA_ET02 )
   END_RUNG wire#w1
   // the same network as SCL:
   IF #PALETIZAR_ET02 AND #ErrorControlPedido AND NOT #Ordenes.Operacion_EvacuarPaleta THEN
       #PALETIZAR_ER01 := TRUE;   // SR flip-flop
   END_IF;
   IF #PALETIZAR_ER02 OR #DESCARGA_ET02 THEN #PALETIZAR_ER01 := FALSE; END_IF;
END_REGION

REGION Network 28: ---- Transferencia de Salida de Paleta
   RUNG wire#powerrail
      Contact( #DESCARGA_ET05 )
      I_Contact( #MFinMoverElev )
      wire#w1
      Contact( #Interlock_TELEV.OrdenTELEV_S1 )
      wire#w2
      S_SR(operand := #DESCARGA_ET06, r1 := #ELEV_ET01)
   END_RUNG
   RUNG wire#w1
      Contact( #Interlock_TELEV.OrdenTELEV_S3 )
   END_RUNG wire#w2
   // the same network as SCL:
   IF #DESCARGA_ET05 AND NOT #MFinMoverElev AND (#Interlock_TELEV.OrdenTELEV_S1 OR #Interlock_TELEV.OrdenTELEV_S3) THEN
       #DESCARGA_ET06 := TRUE;   // SR flip-flop
   END_IF;
   IF #ELEV_ET01 THEN #DESCARGA_ET06 := FALSE; END_IF;
END_REGION

REGION Network 29: ----
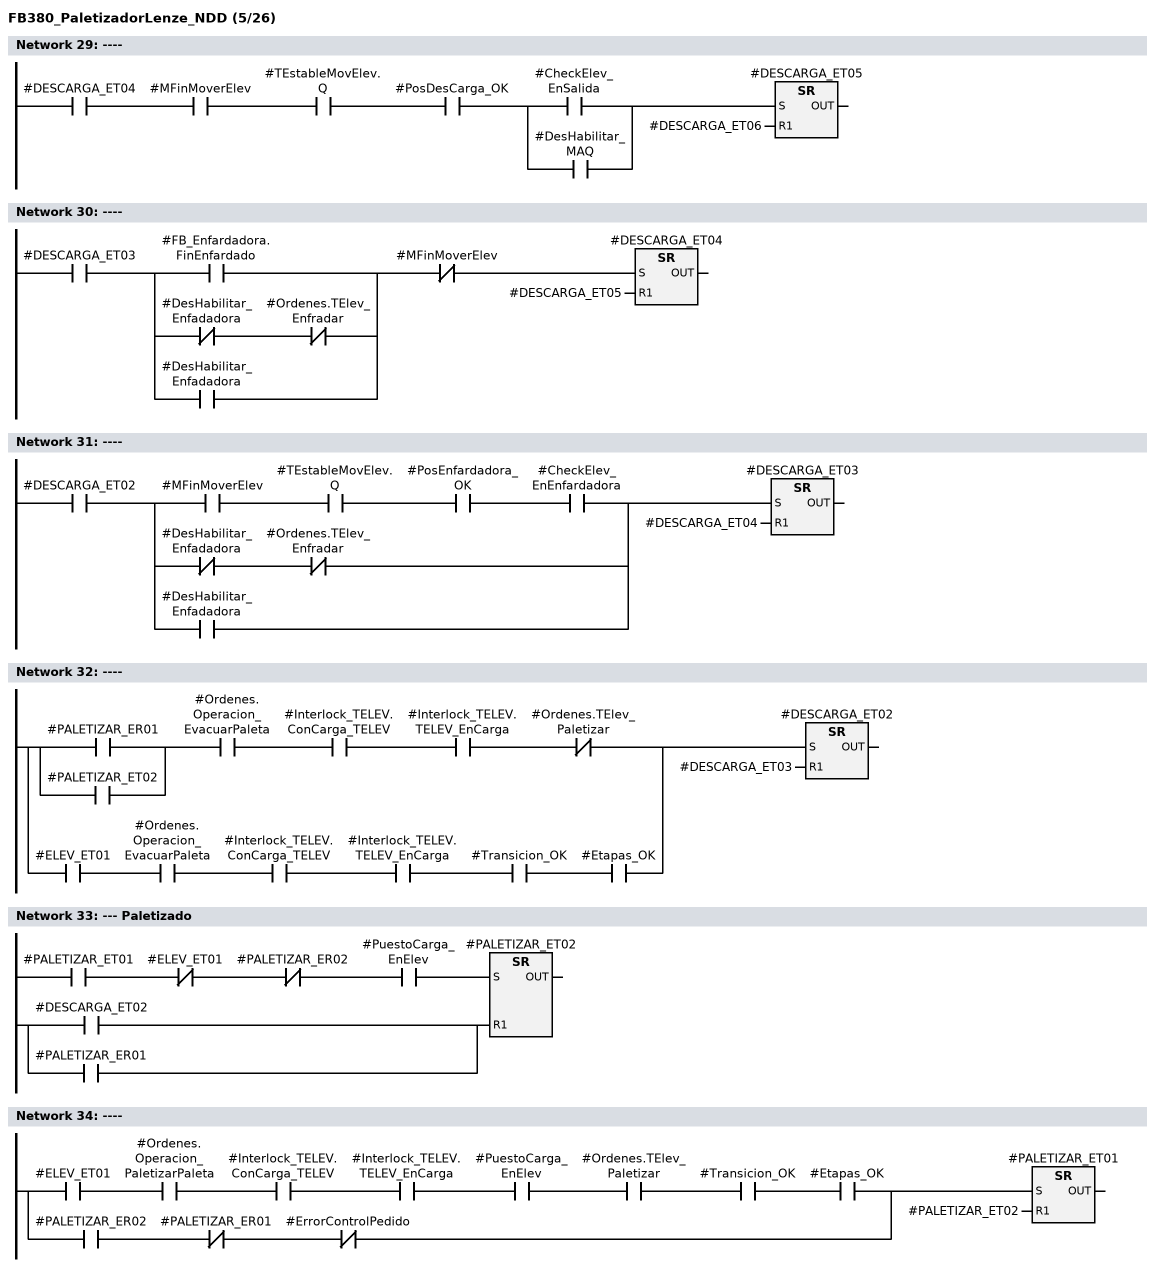
   RUNG wire#powerrail
      Contact( #DESCARGA_ET04 )
      Contact( #MFinMoverElev )
      Contact( #TEstableMovElev.Q )
      Contact( #PosDesCarga_OK )
      wire#w1
      Contact( #CheckElev_EnSalida )
      wire#w2
      S_SR(operand := #DESCARGA_ET05, r1 := #DESCARGA_ET06)
   END_RUNG
   RUNG wire#w1
      Contact( #DesHabilitar_MAQ )
   END_RUNG wire#w2
   // the same network as SCL:
   IF #DESCARGA_ET04 AND #MFinMoverElev AND #TEstableMovElev.Q AND #PosDesCarga_OK AND (#CheckElev_EnSalida OR #DesHabilitar_MAQ) THEN
       #DESCARGA_ET05 := TRUE;   // SR flip-flop
   END_IF;
   IF #DESCARGA_ET06 THEN #DESCARGA_ET05 := FALSE; END_IF;
END_REGION

REGION Network 30: ----
   RUNG wire#powerrail
      Contact( #DESCARGA_ET03 )
      wire#w1
      Contact( #FB_Enfardadora.FinEnfardado )
      wire#w2
      I_Contact( #MFinMoverElev )
      S_SR(operand := #DESCARGA_ET04, r1 := #DESCARGA_ET05)
   END_RUNG
   RUNG wire#w1
      I_Contact( #DesHabilitar_Enfadadora )
      I_Contact( #Ordenes.TElev_Enfradar )
   END_RUNG wire#w2
   RUNG wire#w1
      Contact( #DesHabilitar_Enfadadora )
   END_RUNG wire#w2
   // the same network as SCL:
   IF #DESCARGA_ET03 AND (#FB_Enfardadora.FinEnfardado OR (NOT #DesHabilitar_Enfadadora AND NOT #Ordenes.TElev_Enfradar) OR #DesHabilitar_Enfadadora) AND NOT #MFinMoverElev THEN
       #DESCARGA_ET04 := TRUE;   // SR flip-flop
   END_IF;
   IF #DESCARGA_ET05 THEN #DESCARGA_ET04 := FALSE; END_IF;
END_REGION

REGION Network 31: ----
   RUNG wire#powerrail
      Contact( #DESCARGA_ET02 )
      wire#w1
      Contact( #MFinMoverElev )
      Contact( #TEstableMovElev.Q )
      Contact( #PosEnfardadora_OK )
      Contact( #CheckElev_EnEnfardadora )
      wire#w2
      S_SR(operand := #DESCARGA_ET03, r1 := #DESCARGA_ET04)
   END_RUNG
   RUNG wire#w1
      I_Contact( #DesHabilitar_Enfadadora )
      I_Contact( #Ordenes.TElev_Enfradar )
   END_RUNG wire#w2
   RUNG wire#w1
      Contact( #DesHabilitar_Enfadadora )
   END_RUNG wire#w2
   // the same network as SCL:
   IF #DESCARGA_ET02 AND ((#MFinMoverElev AND #TEstableMovElev.Q AND #PosEnfardadora_OK AND #CheckElev_EnEnfardadora) OR (NOT #DesHabilitar_Enfadadora AND NOT #Ordenes.TElev_Enfradar) OR #DesHabilitar_Enfadadora) THEN
       #DESCARGA_ET03 := TRUE;   // SR flip-flop
   END_IF;
   IF #DESCARGA_ET04 THEN #DESCARGA_ET03 := FALSE; END_IF;
END_REGION

REGION Network 32: ----
   RUNG wire#powerrail
      Contact( #PALETIZAR_ER01 )
      wire#w1
      Contact( #Ordenes.Operacion_EvacuarPaleta )
      Contact( #Interlock_TELEV.ConCarga_TELEV )
      Contact( #Interlock_TELEV.TELEV_EnCarga )
      I_Contact( #Ordenes.TElev_Paletizar )
      wire#w2
      S_SR(operand := #DESCARGA_ET02, r1 := #DESCARGA_ET03)
   END_RUNG
   RUNG wire#powerrail
      Contact( #PALETIZAR_ET02 )
   END_RUNG wire#w1
   RUNG wire#powerrail
      Contact( #ELEV_ET01 )
      Contact( #Ordenes.Operacion_EvacuarPaleta )
      Contact( #Interlock_TELEV.ConCarga_TELEV )
      Contact( #Interlock_TELEV.TELEV_EnCarga )
      Contact( #Transicion_OK )
      Contact( #Etapas_OK )
   END_RUNG wire#w2
   // the same network as SCL:
   IF ((#PALETIZAR_ER01 OR #PALETIZAR_ET02) AND #Ordenes.Operacion_EvacuarPaleta AND #Interlock_TELEV.ConCarga_TELEV AND #Interlock_TELEV.TELEV_EnCarga AND NOT #Ordenes.TElev_Paletizar) OR (#ELEV_ET01 AND #Ordenes.Operacion_EvacuarPaleta AND #Interlock_TELEV.ConCarga_TELEV AND #Interlock_TELEV.TELEV_EnCarga AND #Transicion_OK AND #Etapas_OK) THEN
       #DESCARGA_ET02 := TRUE;   // SR flip-flop
   END_IF;
   IF #DESCARGA_ET03 THEN #DESCARGA_ET02 := FALSE; END_IF;
END_REGION

REGION Network 33: --- Paletizado
   RUNG wire#powerrail
      Contact( #PALETIZAR_ET01 )
      I_Contact( #ELEV_ET01 )
      I_Contact( #PALETIZAR_ER02 )
      Contact( #PuestoCarga_EnElev )
      S_SR(operand := #PALETIZAR_ET02, r1 := wire#w1)
   END_RUNG
   RUNG wire#powerrail
      Contact( #DESCARGA_ET02 )
   END_RUNG wire#w1
   RUNG wire#powerrail
      Contact( #PALETIZAR_ER01 )
   END_RUNG wire#w1
   // the same network as SCL:
   IF #PALETIZAR_ET01 AND NOT #ELEV_ET01 AND NOT #PALETIZAR_ER02 AND #PuestoCarga_EnElev THEN
       #PALETIZAR_ET02 := TRUE;   // SR flip-flop
   END_IF;
   IF #DESCARGA_ET02 OR #PALETIZAR_ER01 THEN #PALETIZAR_ET02 := FALSE; END_IF;
END_REGION

REGION Network 34: ----
   RUNG wire#powerrail
      Contact( #ELEV_ET01 )
      Contact( #Ordenes.Operacion_PaletizarPaleta )
      Contact( #Interlock_TELEV.ConCarga_TELEV )
      Contact( #Interlock_TELEV.TELEV_EnCarga )
      Contact( #PuestoCarga_EnElev )
      Contact( #Ordenes.TElev_Paletizar )
      Contact( #Transicion_OK )
      Contact( #Etapas_OK )
      wire#w1
      S_SR(operand := #PALETIZAR_ET01, r1 := #PALETIZAR_ET02)
   END_RUNG
   RUNG wire#powerrail
      Contact( #PALETIZAR_ER02 )
      I_Contact( #PALETIZAR_ER01 )
      I_Contact( #ErrorControlPedido )
   END_RUNG wire#w1
   // the same network as SCL:
   IF (#ELEV_ET01 AND #Ordenes.Operacion_PaletizarPaleta AND #Interlock_TELEV.ConCarga_TELEV AND #Interlock_TELEV.TELEV_EnCarga AND #PuestoCarga_EnElev AND #Ordenes.TElev_Paletizar AND #Transicion_OK AND #Etapas_OK) OR (#PALETIZAR_ER02 AND NOT #PALETIZAR_ER01 AND NOT #ErrorControlPedido) THEN
       #PALETIZAR_ET01 := TRUE;   // SR flip-flop
   END_IF;
   IF #PALETIZAR_ET02 THEN #PALETIZAR_ET01 := FALSE; END_IF;
END_REGION

REGION Network 35: ---- Orden de Transferencia del Elevador a la Horquilla
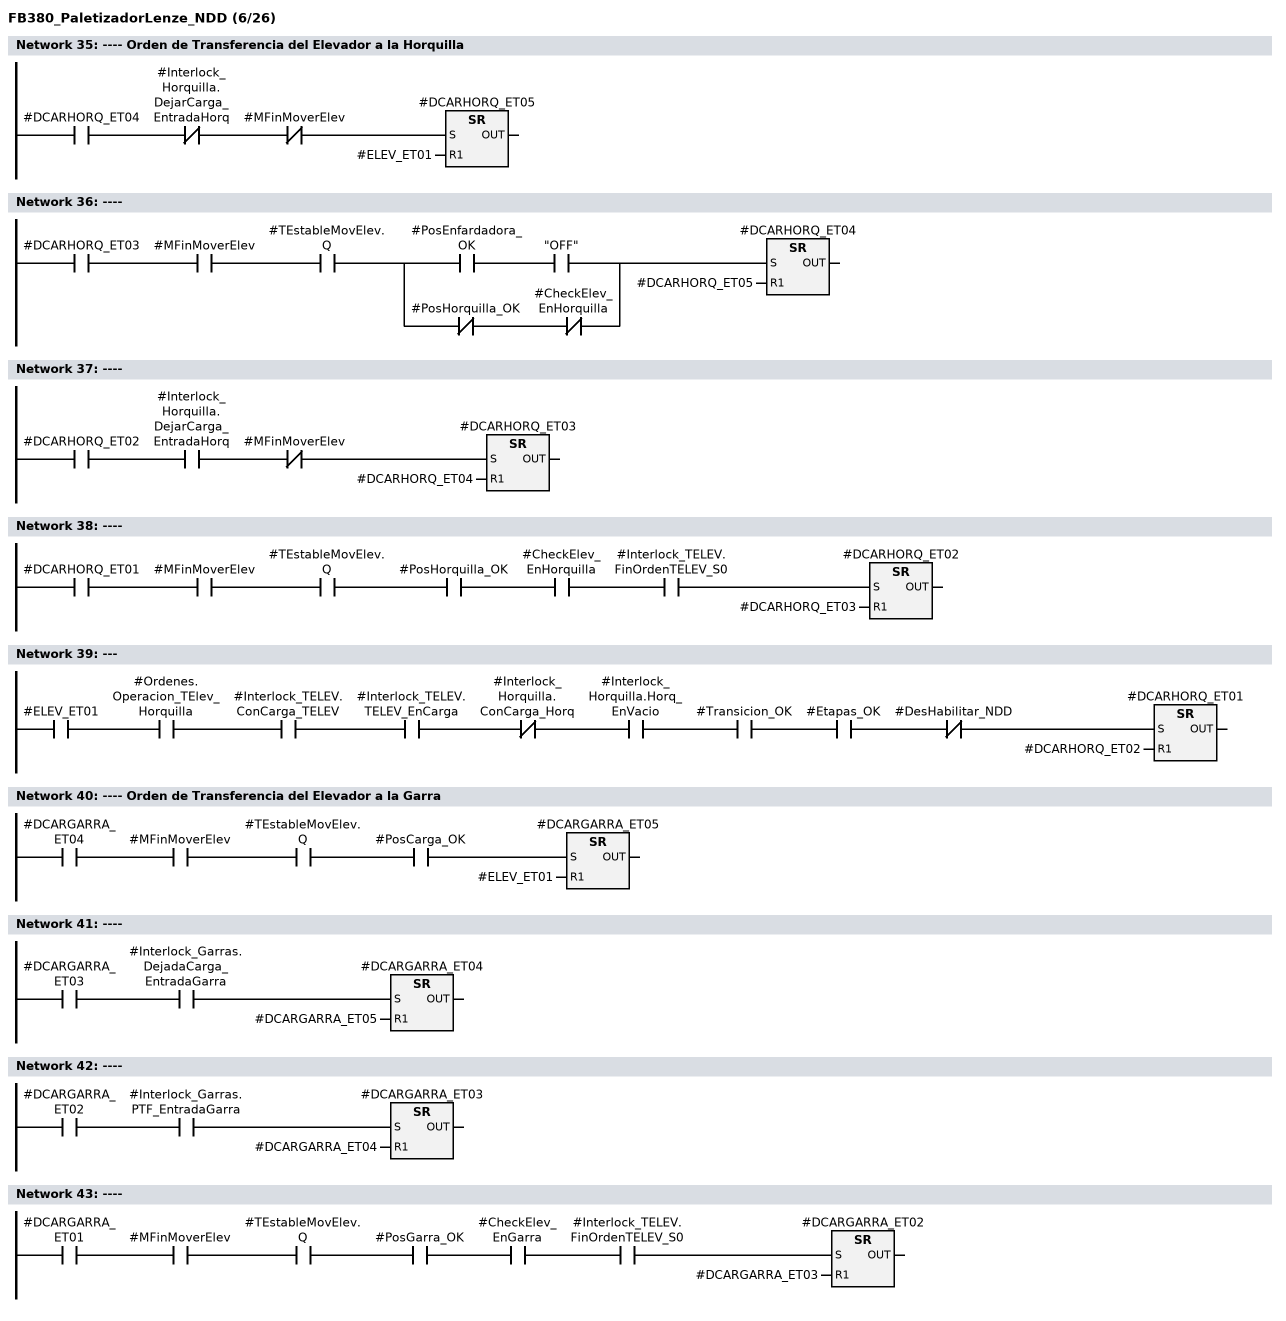
   RUNG wire#powerrail
      Contact( #DCARHORQ_ET04 )
      I_Contact( #Interlock_Horquilla.DejarCarga_EntradaHorq )
      I_Contact( #MFinMoverElev )
      S_SR(operand := #DCARHORQ_ET05, r1 := #ELEV_ET01)
   END_RUNG
   // the same network as SCL:
   IF #DCARHORQ_ET04 AND NOT #Interlock_Horquilla.DejarCarga_EntradaHorq AND NOT #MFinMoverElev THEN
       #DCARHORQ_ET05 := TRUE;   // SR flip-flop
   END_IF;
   IF #ELEV_ET01 THEN #DCARHORQ_ET05 := FALSE; END_IF;
END_REGION

REGION Network 36: ----
   RUNG wire#powerrail
      Contact( #DCARHORQ_ET03 )
      Contact( #MFinMoverElev )
      Contact( #TEstableMovElev.Q )
      wire#w1
      Contact( #PosEnfardadora_OK )
      Contact( "OFF" )
      wire#w2
      S_SR(operand := #DCARHORQ_ET04, r1 := #DCARHORQ_ET05)
   END_RUNG
   RUNG wire#w1
      I_Contact( #PosHorquilla_OK )
      I_Contact( #CheckElev_EnHorquilla )
   END_RUNG wire#w2
   // the same network as SCL:
   IF #DCARHORQ_ET03 AND #MFinMoverElev AND #TEstableMovElev.Q AND ((#PosEnfardadora_OK AND "OFF") OR (NOT #PosHorquilla_OK AND NOT #CheckElev_EnHorquilla)) THEN
       #DCARHORQ_ET04 := TRUE;   // SR flip-flop
   END_IF;
   IF #DCARHORQ_ET05 THEN #DCARHORQ_ET04 := FALSE; END_IF;
END_REGION

REGION Network 37: ----
   RUNG wire#powerrail
      Contact( #DCARHORQ_ET02 )
      Contact( #Interlock_Horquilla.DejarCarga_EntradaHorq )
      I_Contact( #MFinMoverElev )
      S_SR(operand := #DCARHORQ_ET03, r1 := #DCARHORQ_ET04)
   END_RUNG
   // the same network as SCL:
   IF #DCARHORQ_ET02 AND #Interlock_Horquilla.DejarCarga_EntradaHorq AND NOT #MFinMoverElev THEN
       #DCARHORQ_ET03 := TRUE;   // SR flip-flop
   END_IF;
   IF #DCARHORQ_ET04 THEN #DCARHORQ_ET03 := FALSE; END_IF;
END_REGION

REGION Network 38: ----
   RUNG wire#powerrail
      Contact( #DCARHORQ_ET01 )
      Contact( #MFinMoverElev )
      Contact( #TEstableMovElev.Q )
      Contact( #PosHorquilla_OK )
      Contact( #CheckElev_EnHorquilla )
      Contact( #Interlock_TELEV.FinOrdenTELEV_S0 )
      S_SR(operand := #DCARHORQ_ET02, r1 := #DCARHORQ_ET03)
   END_RUNG
   // the same network as SCL:
   IF #DCARHORQ_ET01 AND #MFinMoverElev AND #TEstableMovElev.Q AND #PosHorquilla_OK AND #CheckElev_EnHorquilla AND #Interlock_TELEV.FinOrdenTELEV_S0 THEN
       #DCARHORQ_ET02 := TRUE;   // SR flip-flop
   END_IF;
   IF #DCARHORQ_ET03 THEN #DCARHORQ_ET02 := FALSE; END_IF;
END_REGION

REGION Network 39: ---
   RUNG wire#powerrail
      Contact( #ELEV_ET01 )
      Contact( #Ordenes.Operacion_TElev_Horquilla )
      Contact( #Interlock_TELEV.ConCarga_TELEV )
      Contact( #Interlock_TELEV.TELEV_EnCarga )
      I_Contact( #Interlock_Horquilla.ConCarga_Horq )
      Contact( #Interlock_Horquilla.Horq_EnVacio )
      Contact( #Transicion_OK )
      Contact( #Etapas_OK )
      I_Contact( #DesHabilitar_NDD )
      S_SR(operand := #DCARHORQ_ET01, r1 := #DCARHORQ_ET02)
   END_RUNG
   // the same network as SCL:
   IF #ELEV_ET01 AND #Ordenes.Operacion_TElev_Horquilla AND #Interlock_TELEV.ConCarga_TELEV AND #Interlock_TELEV.TELEV_EnCarga AND NOT #Interlock_Horquilla.ConCarga_Horq AND #Interlock_Horquilla.Horq_EnVacio AND #Transicion_OK AND #Etapas_OK AND NOT #DesHabilitar_NDD THEN
       #DCARHORQ_ET01 := TRUE;   // SR flip-flop
   END_IF;
   IF #DCARHORQ_ET02 THEN #DCARHORQ_ET01 := FALSE; END_IF;
END_REGION

REGION Network 40: ---- Orden de Transferencia del Elevador a la Garra
   RUNG wire#powerrail
      Contact( #DCARGARRA_ET04 )
      Contact( #MFinMoverElev )
      Contact( #TEstableMovElev.Q )
      Contact( #PosCarga_OK )
      S_SR(operand := #DCARGARRA_ET05, r1 := #ELEV_ET01)
   END_RUNG
   // the same network as SCL:
   IF #DCARGARRA_ET04 AND #MFinMoverElev AND #TEstableMovElev.Q AND #PosCarga_OK THEN
       #DCARGARRA_ET05 := TRUE;   // SR flip-flop
   END_IF;
   IF #ELEV_ET01 THEN #DCARGARRA_ET05 := FALSE; END_IF;
END_REGION

REGION Network 41: ----
   RUNG wire#powerrail
      Contact( #DCARGARRA_ET03 )
      Contact( #Interlock_Garras.DejadaCarga_EntradaGarra )
      S_SR(operand := #DCARGARRA_ET04, r1 := #DCARGARRA_ET05)
   END_RUNG
   // the same network as SCL:
   IF #DCARGARRA_ET03 AND #Interlock_Garras.DejadaCarga_EntradaGarra THEN
       #DCARGARRA_ET04 := TRUE;   // SR flip-flop
   END_IF;
   IF #DCARGARRA_ET05 THEN #DCARGARRA_ET04 := FALSE; END_IF;
END_REGION

REGION Network 42: ----
   RUNG wire#powerrail
      Contact( #DCARGARRA_ET02 )
      Contact( #Interlock_Garras.PTF_EntradaGarra )
      S_SR(operand := #DCARGARRA_ET03, r1 := #DCARGARRA_ET04)
   END_RUNG
   // the same network as SCL:
   IF #DCARGARRA_ET02 AND #Interlock_Garras.PTF_EntradaGarra THEN
       #DCARGARRA_ET03 := TRUE;   // SR flip-flop
   END_IF;
   IF #DCARGARRA_ET04 THEN #DCARGARRA_ET03 := FALSE; END_IF;
END_REGION

REGION Network 43: ----
   RUNG wire#powerrail
      Contact( #DCARGARRA_ET01 )
      Contact( #MFinMoverElev )
      Contact( #TEstableMovElev.Q )
      Contact( #PosGarra_OK )
      Contact( #CheckElev_EnGarra )
      Contact( #Interlock_TELEV.FinOrdenTELEV_S0 )
      S_SR(operand := #DCARGARRA_ET02, r1 := #DCARGARRA_ET03)
   END_RUNG
   // the same network as SCL:
   IF #DCARGARRA_ET01 AND #MFinMoverElev AND #TEstableMovElev.Q AND #PosGarra_OK AND #CheckElev_EnGarra AND #Interlock_TELEV.FinOrdenTELEV_S0 THEN
       #DCARGARRA_ET02 := TRUE;   // SR flip-flop
   END_IF;
   IF #DCARGARRA_ET03 THEN #DCARGARRA_ET02 := FALSE; END_IF;
END_REGION

REGION Network 44: ---
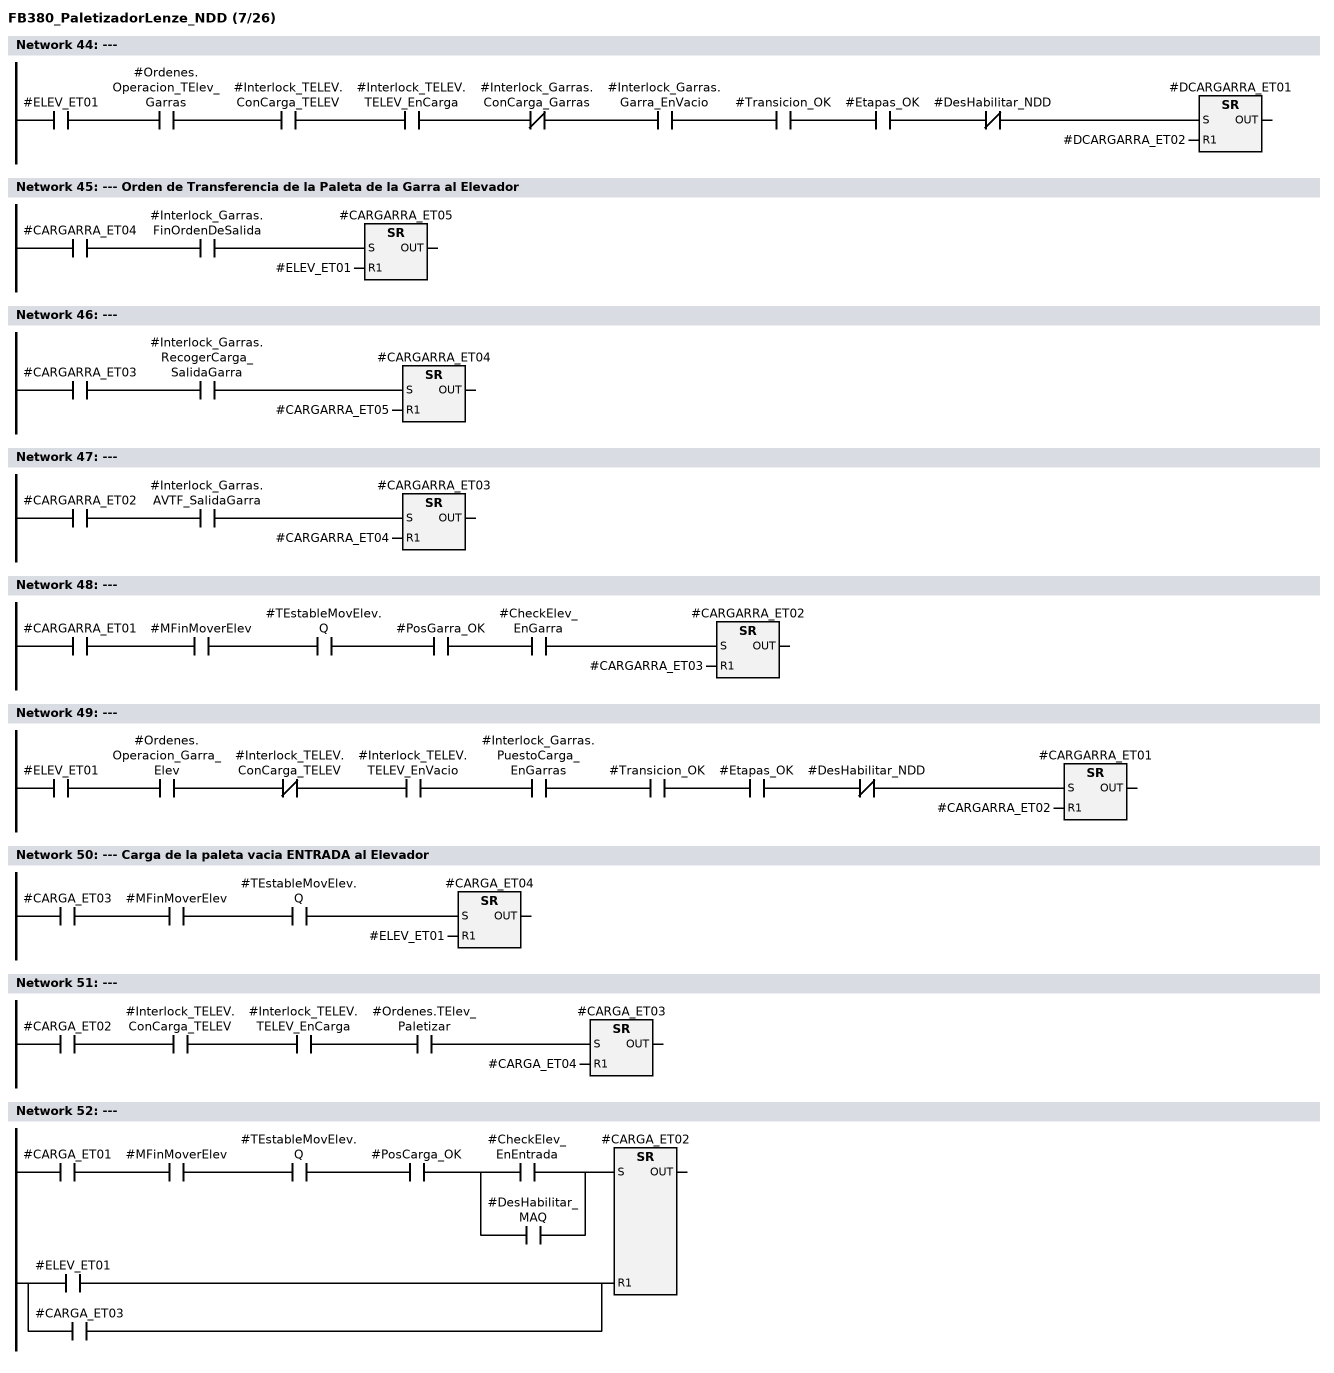
   RUNG wire#powerrail
      Contact( #ELEV_ET01 )
      Contact( #Ordenes.Operacion_TElev_Garras )
      Contact( #Interlock_TELEV.ConCarga_TELEV )
      Contact( #Interlock_TELEV.TELEV_EnCarga )
      I_Contact( #Interlock_Garras.ConCarga_Garras )
      Contact( #Interlock_Garras.Garra_EnVacio )
      Contact( #Transicion_OK )
      Contact( #Etapas_OK )
      I_Contact( #DesHabilitar_NDD )
      S_SR(operand := #DCARGARRA_ET01, r1 := #DCARGARRA_ET02)
   END_RUNG
   // the same network as SCL:
   IF #ELEV_ET01 AND #Ordenes.Operacion_TElev_Garras AND #Interlock_TELEV.ConCarga_TELEV AND #Interlock_TELEV.TELEV_EnCarga AND NOT #Interlock_Garras.ConCarga_Garras AND #Interlock_Garras.Garra_EnVacio AND #Transicion_OK AND #Etapas_OK AND NOT #DesHabilitar_NDD THEN
       #DCARGARRA_ET01 := TRUE;   // SR flip-flop
   END_IF;
   IF #DCARGARRA_ET02 THEN #DCARGARRA_ET01 := FALSE; END_IF;
END_REGION

REGION Network 45: --- Orden de Transferencia de la Paleta de la Garra al Elevador
   RUNG wire#powerrail
      Contact( #CARGARRA_ET04 )
      Contact( #Interlock_Garras.FinOrdenDeSalida )
      S_SR(operand := #CARGARRA_ET05, r1 := #ELEV_ET01)
   END_RUNG
   // the same network as SCL:
   IF #CARGARRA_ET04 AND #Interlock_Garras.FinOrdenDeSalida THEN
       #CARGARRA_ET05 := TRUE;   // SR flip-flop
   END_IF;
   IF #ELEV_ET01 THEN #CARGARRA_ET05 := FALSE; END_IF;
END_REGION

REGION Network 46: ---
   RUNG wire#powerrail
      Contact( #CARGARRA_ET03 )
      Contact( #Interlock_Garras.RecogerCarga_SalidaGarra )
      S_SR(operand := #CARGARRA_ET04, r1 := #CARGARRA_ET05)
   END_RUNG
   // the same network as SCL:
   IF #CARGARRA_ET03 AND #Interlock_Garras.RecogerCarga_SalidaGarra THEN
       #CARGARRA_ET04 := TRUE;   // SR flip-flop
   END_IF;
   IF #CARGARRA_ET05 THEN #CARGARRA_ET04 := FALSE; END_IF;
END_REGION

REGION Network 47: ---
   RUNG wire#powerrail
      Contact( #CARGARRA_ET02 )
      Contact( #Interlock_Garras.AVTF_SalidaGarra )
      S_SR(operand := #CARGARRA_ET03, r1 := #CARGARRA_ET04)
   END_RUNG
   // the same network as SCL:
   IF #CARGARRA_ET02 AND #Interlock_Garras.AVTF_SalidaGarra THEN
       #CARGARRA_ET03 := TRUE;   // SR flip-flop
   END_IF;
   IF #CARGARRA_ET04 THEN #CARGARRA_ET03 := FALSE; END_IF;
END_REGION

REGION Network 48: ---
   RUNG wire#powerrail
      Contact( #CARGARRA_ET01 )
      Contact( #MFinMoverElev )
      Contact( #TEstableMovElev.Q )
      Contact( #PosGarra_OK )
      Contact( #CheckElev_EnGarra )
      S_SR(operand := #CARGARRA_ET02, r1 := #CARGARRA_ET03)
   END_RUNG
   // the same network as SCL:
   IF #CARGARRA_ET01 AND #MFinMoverElev AND #TEstableMovElev.Q AND #PosGarra_OK AND #CheckElev_EnGarra THEN
       #CARGARRA_ET02 := TRUE;   // SR flip-flop
   END_IF;
   IF #CARGARRA_ET03 THEN #CARGARRA_ET02 := FALSE; END_IF;
END_REGION

REGION Network 49: ---
   RUNG wire#powerrail
      Contact( #ELEV_ET01 )
      Contact( #Ordenes.Operacion_Garra_Elev )
      I_Contact( #Interlock_TELEV.ConCarga_TELEV )
      Contact( #Interlock_TELEV.TELEV_EnVacio )
      Contact( #Interlock_Garras.PuestoCarga_EnGarras )
      Contact( #Transicion_OK )
      Contact( #Etapas_OK )
      I_Contact( #DesHabilitar_NDD )
      S_SR(operand := #CARGARRA_ET01, r1 := #CARGARRA_ET02)
   END_RUNG
   // the same network as SCL:
   IF #ELEV_ET01 AND #Ordenes.Operacion_Garra_Elev AND NOT #Interlock_TELEV.ConCarga_TELEV AND #Interlock_TELEV.TELEV_EnVacio AND #Interlock_Garras.PuestoCarga_EnGarras AND #Transicion_OK AND #Etapas_OK AND NOT #DesHabilitar_NDD THEN
       #CARGARRA_ET01 := TRUE;   // SR flip-flop
   END_IF;
   IF #CARGARRA_ET02 THEN #CARGARRA_ET01 := FALSE; END_IF;
END_REGION

REGION Network 50: --- Carga de la paleta vacia ENTRADA al Elevador
   RUNG wire#powerrail
      Contact( #CARGA_ET03 )
      Contact( #MFinMoverElev )
      Contact( #TEstableMovElev.Q )
      S_SR(operand := #CARGA_ET04, r1 := #ELEV_ET01)
   END_RUNG
   // the same network as SCL:
   IF #CARGA_ET03 AND #MFinMoverElev AND #TEstableMovElev.Q THEN
       #CARGA_ET04 := TRUE;   // SR flip-flop
   END_IF;
   IF #ELEV_ET01 THEN #CARGA_ET04 := FALSE; END_IF;
END_REGION

REGION Network 51: ---
   RUNG wire#powerrail
      Contact( #CARGA_ET02 )
      Contact( #Interlock_TELEV.ConCarga_TELEV )
      Contact( #Interlock_TELEV.TELEV_EnCarga )
      Contact( #Ordenes.TElev_Paletizar )
      S_SR(operand := #CARGA_ET03, r1 := #CARGA_ET04)
   END_RUNG
   // the same network as SCL:
   IF #CARGA_ET02 AND #Interlock_TELEV.ConCarga_TELEV AND #Interlock_TELEV.TELEV_EnCarga AND #Ordenes.TElev_Paletizar THEN
       #CARGA_ET03 := TRUE;   // SR flip-flop
   END_IF;
   IF #CARGA_ET04 THEN #CARGA_ET03 := FALSE; END_IF;
END_REGION

REGION Network 52: ---
   RUNG wire#powerrail
      Contact( #CARGA_ET01 )
      Contact( #MFinMoverElev )
      Contact( #TEstableMovElev.Q )
      Contact( #PosCarga_OK )
      wire#w1
      Contact( #CheckElev_EnEntrada )
      wire#w2
      S_SR(operand := #CARGA_ET02, r1 := wire#w3)
   END_RUNG
   RUNG wire#w1
      Contact( #DesHabilitar_MAQ )
   END_RUNG wire#w2
   RUNG wire#powerrail
      Contact( #ELEV_ET01 )
   END_RUNG wire#w3
   RUNG wire#powerrail
      Contact( #CARGA_ET03 )
   END_RUNG wire#w3
   // the same network as SCL:
   IF #CARGA_ET01 AND #MFinMoverElev AND #TEstableMovElev.Q AND #PosCarga_OK AND (#CheckElev_EnEntrada OR #DesHabilitar_MAQ) THEN
       #CARGA_ET02 := TRUE;   // SR flip-flop
   END_IF;
   IF #ELEV_ET01 OR #CARGA_ET03 THEN #CARGA_ET02 := FALSE; END_IF;
END_REGION

REGION Network 53: ---
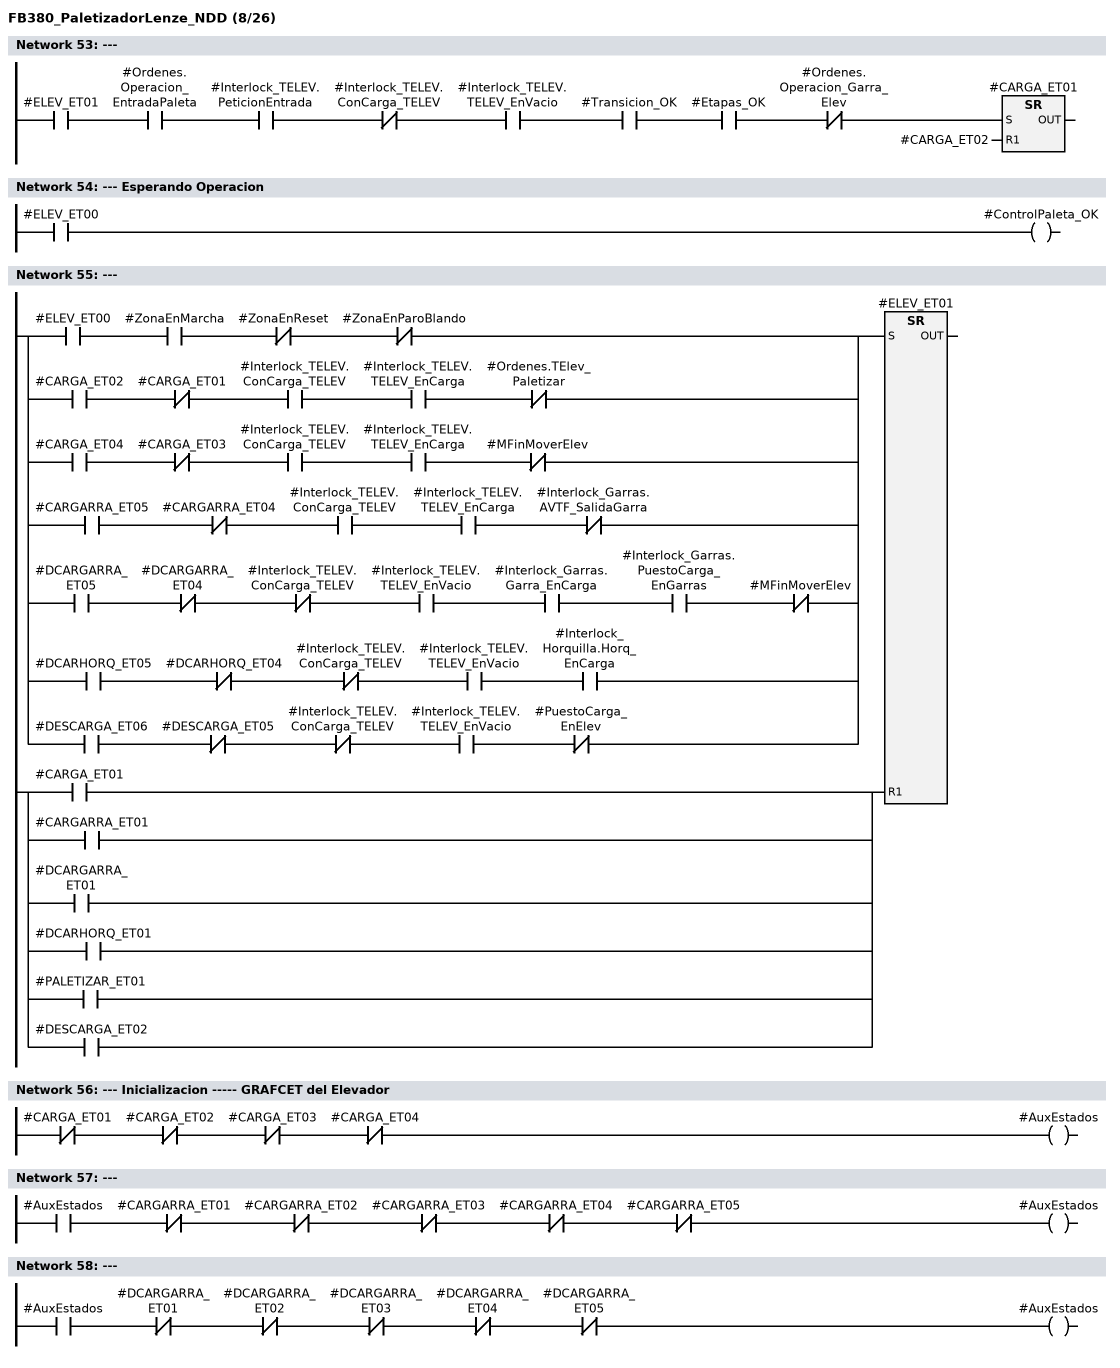
   RUNG wire#powerrail
      Contact( #ELEV_ET01 )
      Contact( #Ordenes.Operacion_EntradaPaleta )
      Contact( #Interlock_TELEV.PeticionEntrada )
      I_Contact( #Interlock_TELEV.ConCarga_TELEV )
      Contact( #Interlock_TELEV.TELEV_EnVacio )
      Contact( #Transicion_OK )
      Contact( #Etapas_OK )
      I_Contact( #Ordenes.Operacion_Garra_Elev )
      S_SR(operand := #CARGA_ET01, r1 := #CARGA_ET02)
   END_RUNG
   // the same network as SCL:
   IF #ELEV_ET01 AND #Ordenes.Operacion_EntradaPaleta AND #Interlock_TELEV.PeticionEntrada AND NOT #Interlock_TELEV.ConCarga_TELEV AND #Interlock_TELEV.TELEV_EnVacio AND #Transicion_OK AND #Etapas_OK AND NOT #Ordenes.Operacion_Garra_Elev THEN
       #CARGA_ET01 := TRUE;   // SR flip-flop
   END_IF;
   IF #CARGA_ET02 THEN #CARGA_ET01 := FALSE; END_IF;
END_REGION

REGION Network 54: --- Esperando Operacion
   RUNG wire#powerrail
      Contact( #ELEV_ET00 )
      Coil( #ControlPaleta_OK )
   END_RUNG
   // the same network as SCL:
   #ControlPaleta_OK := #ELEV_ET00;
END_REGION

REGION Network 55: ---
   RUNG wire#powerrail
      Contact( #ELEV_ET00 )
      Contact( #ZonaEnMarcha )
      I_Contact( #ZonaEnReset )
      I_Contact( #ZonaEnParoBlando )
      wire#w1
      S_SR(operand := #ELEV_ET01, r1 := wire#w2)
   END_RUNG
   RUNG wire#powerrail
      Contact( #CARGA_ET02 )
      I_Contact( #CARGA_ET01 )
      Contact( #Interlock_TELEV.ConCarga_TELEV )
      Contact( #Interlock_TELEV.TELEV_EnCarga )
      I_Contact( #Ordenes.TElev_Paletizar )
   END_RUNG wire#w1
   RUNG wire#powerrail
      Contact( #CARGA_ET04 )
      I_Contact( #CARGA_ET03 )
      Contact( #Interlock_TELEV.ConCarga_TELEV )
      Contact( #Interlock_TELEV.TELEV_EnCarga )
      I_Contact( #MFinMoverElev )
   END_RUNG wire#w1
   RUNG wire#powerrail
      Contact( #CARGARRA_ET05 )
      I_Contact( #CARGARRA_ET04 )
      Contact( #Interlock_TELEV.ConCarga_TELEV )
      Contact( #Interlock_TELEV.TELEV_EnCarga )
      I_Contact( #Interlock_Garras.AVTF_SalidaGarra )
   END_RUNG wire#w1
   RUNG wire#powerrail
      Contact( #DCARGARRA_ET05 )
      I_Contact( #DCARGARRA_ET04 )
      I_Contact( #Interlock_TELEV.ConCarga_TELEV )
      Contact( #Interlock_TELEV.TELEV_EnVacio )
      Contact( #Interlock_Garras.Garra_EnCarga )
      Contact( #Interlock_Garras.PuestoCarga_EnGarras )
      I_Contact( #MFinMoverElev )
   END_RUNG wire#w1
   RUNG wire#powerrail
      Contact( #DCARHORQ_ET05 )
      I_Contact( #DCARHORQ_ET04 )
      I_Contact( #Interlock_TELEV.ConCarga_TELEV )
      Contact( #Interlock_TELEV.TELEV_EnVacio )
      Contact( #Interlock_Horquilla.Horq_EnCarga )
   END_RUNG wire#w1
   RUNG wire#powerrail
      Contact( #DESCARGA_ET06 )
      I_Contact( #DESCARGA_ET05 )
      I_Contact( #Interlock_TELEV.ConCarga_TELEV )
      Contact( #Interlock_TELEV.TELEV_EnVacio )
      I_Contact( #PuestoCarga_EnElev )
   END_RUNG wire#w1
   RUNG wire#powerrail
      Contact( #CARGA_ET01 )
   END_RUNG wire#w2
   RUNG wire#powerrail
      Contact( #CARGARRA_ET01 )
   END_RUNG wire#w2
   RUNG wire#powerrail
      Contact( #DCARGARRA_ET01 )
   END_RUNG wire#w2
   RUNG wire#powerrail
      Contact( #DCARHORQ_ET01 )
   END_RUNG wire#w2
   RUNG wire#powerrail
      Contact( #PALETIZAR_ET01 )
   END_RUNG wire#w2
   RUNG wire#powerrail
      Contact( #DESCARGA_ET02 )
   END_RUNG wire#w2
   // the same network as SCL:
   IF (#ELEV_ET00 AND #ZonaEnMarcha AND NOT #ZonaEnReset AND NOT #ZonaEnParoBlando) OR (#CARGA_ET02 AND NOT #CARGA_ET01 AND #Interlock_TELEV.ConCarga_TELEV AND #Interlock_TELEV.TELEV_EnCarga AND NOT #Ordenes.TElev_Paletizar) OR (#CARGA_ET04 AND NOT #CARGA_ET03 AND #Interlock_TELEV.ConCarga_TELEV AND #Interlock_TELEV.TELEV_EnCarga AND NOT #MFinMoverElev) OR (#CARGARRA_ET05 AND NOT #CARGARRA_ET04 AND #Interlock_TELEV.ConCarga_TELEV AND #Interlock_TELEV.TELEV_EnCarga AND NOT #Interlock_Garras.AVTF_SalidaGarra) OR (#DCARGARRA_ET05 AND NOT #DCARGARRA_ET04 AND NOT #Interlock_TELEV.ConCarga_TELEV AND #Interlock_TELEV.TELEV_EnVacio AND #Interlock_Garras.Garra_EnCarga AND #Interlock_Garras.PuestoCarga_EnGarras AND NOT #MFinMoverElev) OR (#DCARHORQ_ET05 AND NOT #DCARHORQ_ET04 AND NOT #Interlock_TELEV.ConCarga_TELEV AND #Interlock_TELEV.TELEV_EnVacio AND #Interlock_Horquilla.Horq_EnCarga) OR (#DESCARGA_ET06 AND NOT #DESCARGA_ET05 AND NOT #Interlock_TELEV.ConCarga_TELEV AND #Interlock_TELEV.TELEV_EnVacio AND NOT #PuestoCarga_EnElev) THEN
       #ELEV_ET01 := TRUE;   // SR flip-flop
   END_IF;
   IF #CARGA_ET01 OR #CARGARRA_ET01 OR #DCARGARRA_ET01 OR #DCARHORQ_ET01 OR #PALETIZAR_ET01 OR #DESCARGA_ET02 THEN
       #ELEV_ET01 := FALSE;
   END_IF;
END_REGION

REGION Network 56: --- Inicializacion ----- GRAFCET del Elevador
   RUNG wire#powerrail
      I_Contact( #CARGA_ET01 )
      I_Contact( #CARGA_ET02 )
      I_Contact( #CARGA_ET03 )
      I_Contact( #CARGA_ET04 )
      Coil( #AuxEstados )
   END_RUNG
   // the same network as SCL:
   #AuxEstados := NOT #CARGA_ET01 AND NOT #CARGA_ET02 AND NOT #CARGA_ET03 AND NOT #CARGA_ET04;
END_REGION

REGION Network 57: ---
   RUNG wire#powerrail
      Contact( #AuxEstados )
      I_Contact( #CARGARRA_ET01 )
      I_Contact( #CARGARRA_ET02 )
      I_Contact( #CARGARRA_ET03 )
      I_Contact( #CARGARRA_ET04 )
      I_Contact( #CARGARRA_ET05 )
      Coil( #AuxEstados )
   END_RUNG
   // the same network as SCL:
   #AuxEstados := #AuxEstados AND NOT #CARGARRA_ET01 AND NOT #CARGARRA_ET02 AND NOT #CARGARRA_ET03 AND NOT #CARGARRA_ET04 AND NOT #CARGARRA_ET05;
END_REGION

REGION Network 58: ---
   RUNG wire#powerrail
      Contact( #AuxEstados )
      I_Contact( #DCARGARRA_ET01 )
      I_Contact( #DCARGARRA_ET02 )
      I_Contact( #DCARGARRA_ET03 )
      I_Contact( #DCARGARRA_ET04 )
      I_Contact( #DCARGARRA_ET05 )
      Coil( #AuxEstados )
   END_RUNG
   // the same network as SCL:
   #AuxEstados := #AuxEstados AND NOT #DCARGARRA_ET01 AND NOT #DCARGARRA_ET02 AND NOT #DCARGARRA_ET03 AND NOT #DCARGARRA_ET04 AND NOT #DCARGARRA_ET05;
END_REGION

REGION Network 59: ---
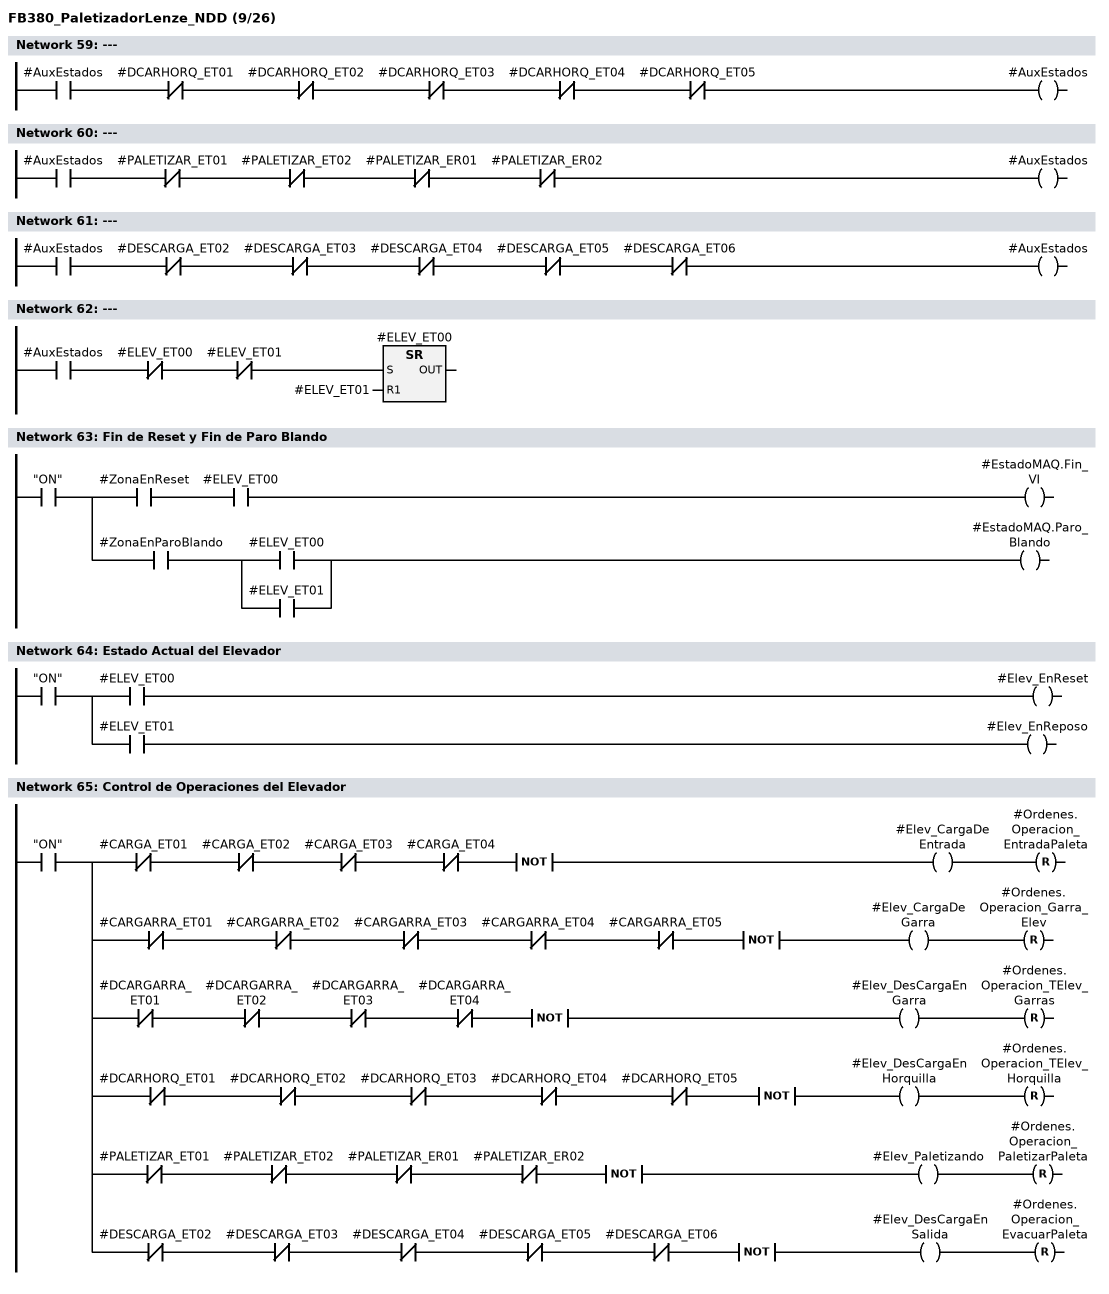
   RUNG wire#powerrail
      Contact( #AuxEstados )
      I_Contact( #DCARHORQ_ET01 )
      I_Contact( #DCARHORQ_ET02 )
      I_Contact( #DCARHORQ_ET03 )
      I_Contact( #DCARHORQ_ET04 )
      I_Contact( #DCARHORQ_ET05 )
      Coil( #AuxEstados )
   END_RUNG
   // the same network as SCL:
   #AuxEstados := #AuxEstados AND NOT #DCARHORQ_ET01 AND NOT #DCARHORQ_ET02 AND NOT #DCARHORQ_ET03 AND NOT #DCARHORQ_ET04 AND NOT #DCARHORQ_ET05;
END_REGION

REGION Network 60: ---
   RUNG wire#powerrail
      Contact( #AuxEstados )
      I_Contact( #PALETIZAR_ET01 )
      I_Contact( #PALETIZAR_ET02 )
      I_Contact( #PALETIZAR_ER01 )
      I_Contact( #PALETIZAR_ER02 )
      Coil( #AuxEstados )
   END_RUNG
   // the same network as SCL:
   #AuxEstados := #AuxEstados AND NOT #PALETIZAR_ET01 AND NOT #PALETIZAR_ET02 AND NOT #PALETIZAR_ER01 AND NOT #PALETIZAR_ER02;
END_REGION

REGION Network 61: ---
   RUNG wire#powerrail
      Contact( #AuxEstados )
      I_Contact( #DESCARGA_ET02 )
      I_Contact( #DESCARGA_ET03 )
      I_Contact( #DESCARGA_ET04 )
      I_Contact( #DESCARGA_ET05 )
      I_Contact( #DESCARGA_ET06 )
      Coil( #AuxEstados )
   END_RUNG
   // the same network as SCL:
   #AuxEstados := #AuxEstados AND NOT #DESCARGA_ET02 AND NOT #DESCARGA_ET03 AND NOT #DESCARGA_ET04 AND NOT #DESCARGA_ET05 AND NOT #DESCARGA_ET06;
END_REGION

REGION Network 62: ---
   RUNG wire#powerrail
      Contact( #AuxEstados )
      I_Contact( #ELEV_ET00 )
      I_Contact( #ELEV_ET01 )
      S_SR(operand := #ELEV_ET00, r1 := #ELEV_ET01)
   END_RUNG
   // the same network as SCL:
   IF #AuxEstados AND NOT #ELEV_ET00 AND NOT #ELEV_ET01 THEN
       #ELEV_ET00 := TRUE;   // SR flip-flop
   END_IF;
   IF #ELEV_ET01 THEN #ELEV_ET00 := FALSE; END_IF;
END_REGION

REGION Network 63: Fin de Reset y Fin de Paro Blando
   RUNG wire#powerrail
      Contact( "ON" )
      wire#w1
      Contact( #ZonaEnReset )
      Contact( #ELEV_ET00 )
      Coil( #EstadoMAQ.Fin_VI )
   END_RUNG
   RUNG wire#w1
      Contact( #ZonaEnParoBlando )
      wire#w2
      Contact( #ELEV_ET00 )
      wire#w3
      Coil( #EstadoMAQ.Paro_Blando )
   END_RUNG
   RUNG wire#w2
      Contact( #ELEV_ET01 )
   END_RUNG wire#w3
   // the same network as SCL:
   #EstadoMAQ.Fin_VI := "ON" AND #ZonaEnReset AND #ELEV_ET00;
   #EstadoMAQ.Paro_Blando := "ON" AND #ZonaEnParoBlando AND (#ELEV_ET00 OR #ELEV_ET01);
END_REGION

REGION Network 64: Estado Actual del Elevador
   RUNG wire#powerrail
      Contact( "ON" )
      wire#w1
      Contact( #ELEV_ET00 )
      Coil( #Elev_EnReset )
   END_RUNG
   RUNG wire#w1
      Contact( #ELEV_ET01 )
      Coil( #Elev_EnReposo )
   END_RUNG
   // the same network as SCL:
   #Elev_EnReset := "ON" AND #ELEV_ET00;
   #Elev_EnReposo := "ON" AND #ELEV_ET01;
END_REGION

REGION Network 65: Control de Operaciones del Elevador
   RUNG wire#powerrail
      Contact( "ON" )
      wire#w1
      I_Contact( #CARGA_ET01 )
      I_Contact( #CARGA_ET02 )
      I_Contact( #CARGA_ET03 )
      I_Contact( #CARGA_ET04 )
      Not()
      Coil( #Elev_CargaDeEntrada )
      R_Coil( #Ordenes.Operacion_EntradaPaleta )
   END_RUNG
   RUNG wire#w1
      I_Contact( #CARGARRA_ET01 )
      I_Contact( #CARGARRA_ET02 )
      I_Contact( #CARGARRA_ET03 )
      I_Contact( #CARGARRA_ET04 )
      I_Contact( #CARGARRA_ET05 )
      Not()
      Coil( #Elev_CargaDeGarra )
      R_Coil( #Ordenes.Operacion_Garra_Elev )
   END_RUNG
   RUNG wire#w1
      I_Contact( #DCARGARRA_ET01 )
      I_Contact( #DCARGARRA_ET02 )
      I_Contact( #DCARGARRA_ET03 )
      I_Contact( #DCARGARRA_ET04 )
      Not()
      Coil( #Elev_DesCargaEnGarra )
      R_Coil( #Ordenes.Operacion_TElev_Garras )
   END_RUNG
   RUNG wire#w1
      I_Contact( #DCARHORQ_ET01 )
      I_Contact( #DCARHORQ_ET02 )
      I_Contact( #DCARHORQ_ET03 )
      I_Contact( #DCARHORQ_ET04 )
      I_Contact( #DCARHORQ_ET05 )
      Not()
      Coil( #Elev_DesCargaEnHorquilla )
      R_Coil( #Ordenes.Operacion_TElev_Horquilla )
   END_RUNG
   RUNG wire#w1
      I_Contact( #PALETIZAR_ET01 )
      I_Contact( #PALETIZAR_ET02 )
      I_Contact( #PALETIZAR_ER01 )
      I_Contact( #PALETIZAR_ER02 )
      Not()
      Coil( #Elev_Paletizando )
      R_Coil( #Ordenes.Operacion_PaletizarPaleta )
   END_RUNG
   RUNG wire#w1
      I_Contact( #DESCARGA_ET02 )
      I_Contact( #DESCARGA_ET03 )
      I_Contact( #DESCARGA_ET04 )
      I_Contact( #DESCARGA_ET05 )
      I_Contact( #DESCARGA_ET06 )
      Not()
      Coil( #Elev_DesCargaEnSalida )
      R_Coil( #Ordenes.Operacion_EvacuarPaleta )
   END_RUNG
   // the same network as SCL:
   #Elev_CargaDeEntrada := NOT ("ON" AND NOT #CARGA_ET01 AND NOT #CARGA_ET02 AND NOT #CARGA_ET03 AND NOT #CARGA_ET04);
   IF #Elev_CargaDeEntrada THEN #Ordenes.Operacion_EntradaPaleta := FALSE; END_IF;
   #Elev_CargaDeGarra := NOT ("ON" AND NOT #CARGARRA_ET01 AND NOT #CARGARRA_ET02 AND NOT #CARGARRA_ET03 AND NOT #CARGARRA_ET04 AND NOT #CARGARRA_ET05);
   IF #Elev_CargaDeGarra THEN #Ordenes.Operacion_Garra_Elev := FALSE; END_IF;
   #Elev_DesCargaEnGarra := NOT ("ON" AND NOT #DCARGARRA_ET01 AND NOT #DCARGARRA_ET02 AND NOT #DCARGARRA_ET03 AND NOT #DCARGARRA_ET04);
   IF #Elev_DesCargaEnGarra THEN #Ordenes.Operacion_TElev_Garras := FALSE; END_IF;
   #Elev_DesCargaEnHorquilla := NOT ("ON" AND NOT #DCARHORQ_ET01 AND NOT #DCARHORQ_ET02 AND NOT #DCARHORQ_ET03 AND NOT #DCARHORQ_ET04 AND NOT #DCARHORQ_ET05);
   IF #Elev_DesCargaEnHorquilla THEN #Ordenes.Operacion_TElev_Horquilla := FALSE; END_IF;
   #Elev_Paletizando := NOT ("ON" AND NOT #PALETIZAR_ET01 AND NOT #PALETIZAR_ET02 AND NOT #PALETIZAR_ER01 AND NOT #PALETIZAR_ER02);
   IF #Elev_Paletizando THEN #Ordenes.Operacion_PaletizarPaleta := FALSE; END_IF;
   #Elev_DesCargaEnSalida := NOT ("ON" AND NOT #DESCARGA_ET02 AND NOT #DESCARGA_ET03 AND NOT #DESCARGA_ET04 AND NOT #DESCARGA_ET05 AND NOT #DESCARGA_ET06);
   IF #Elev_DesCargaEnSalida THEN #Ordenes.Operacion_EvacuarPaleta := FALSE; END_IF;
END_REGION

REGION Network 66: Control de la Operacion de Horquilla con Garra
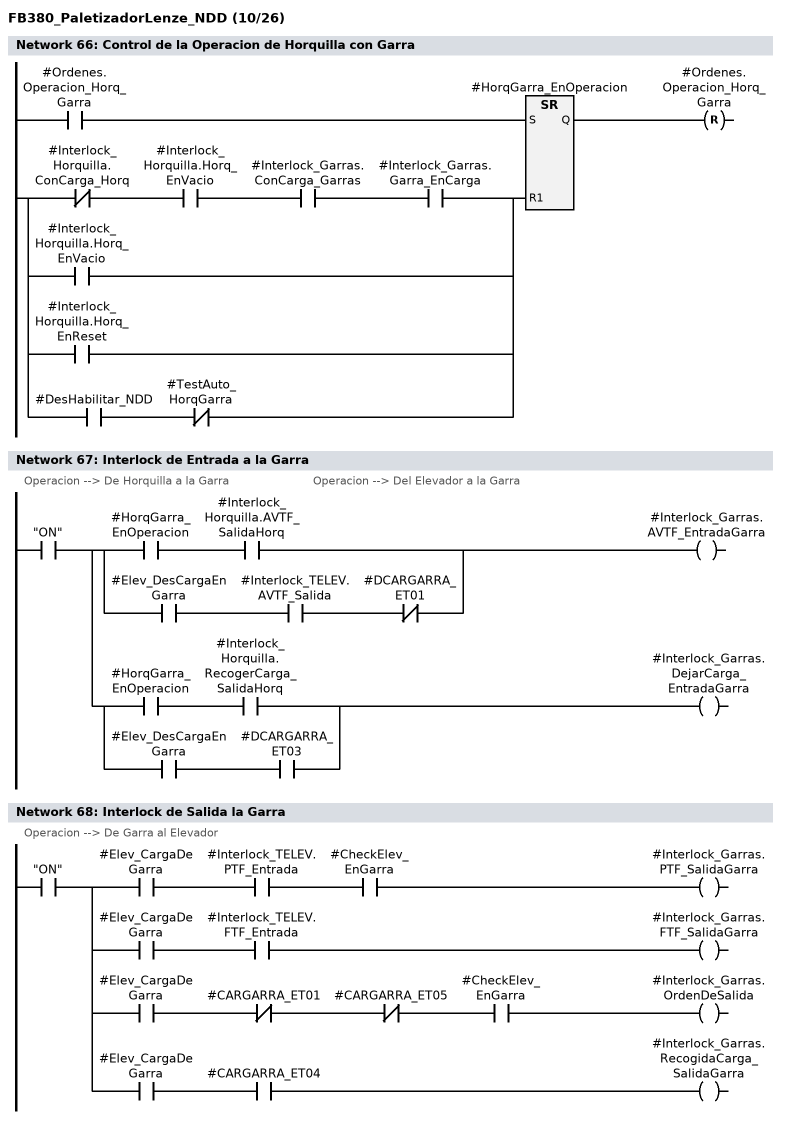
   RUNG wire#powerrail
      Contact( #Ordenes.Operacion_Horq_Garra )
      S_SR(operand := #HorqGarra_EnOperacion, r1 := wire#w1)
      R_Coil( #Ordenes.Operacion_Horq_Garra )
   END_RUNG
   RUNG wire#powerrail
      I_Contact( #Interlock_Horquilla.ConCarga_Horq )
      Contact( #Interlock_Horquilla.Horq_EnVacio )
      Contact( #Interlock_Garras.ConCarga_Garras )
      Contact( #Interlock_Garras.Garra_EnCarga )
   END_RUNG wire#w1
   RUNG wire#powerrail
      Contact( #Interlock_Horquilla.Horq_EnVacio )
   END_RUNG wire#w1
   RUNG wire#powerrail
      Contact( #Interlock_Horquilla.Horq_EnReset )
   END_RUNG wire#w1
   RUNG wire#powerrail
      Contact( #DesHabilitar_NDD )
      I_Contact( #TestAuto_HorqGarra )
   END_RUNG wire#w1
   // the same network as SCL:
   IF #Ordenes.Operacion_Horq_Garra THEN
       #HorqGarra_EnOperacion := TRUE;   // SR flip-flop
   END_IF;
   IF (NOT #Interlock_Horquilla.ConCarga_Horq AND #Interlock_Horquilla.Horq_EnVacio AND #Interlock_Garras.ConCarga_Garras AND #Interlock_Garras.Garra_EnCarga) OR #Interlock_Horquilla.Horq_EnVacio OR #Interlock_Horquilla.Horq_EnReset OR (#DesHabilitar_NDD AND NOT #TestAuto_HorqGarra) THEN
       #HorqGarra_EnOperacion := FALSE;
   END_IF;
   IF #HorqGarra_EnOperacion THEN #Ordenes.Operacion_Horq_Garra := FALSE; END_IF;
END_REGION

REGION Network 67: Interlock de Entrada a la Garra
   // Operacion --> De Horquilla a la Garra                        Operacion --> Del Elevador a la Garra
   RUNG wire#powerrail
      Contact( "ON" )
      wire#w1
      Contact( #HorqGarra_EnOperacion )
      Contact( #Interlock_Horquilla.AVTF_SalidaHorq )
      wire#w2
      Coil( #Interlock_Garras.AVTF_EntradaGarra )
   END_RUNG
   RUNG wire#w1
      Contact( #Elev_DesCargaEnGarra )
      Contact( #Interlock_TELEV.AVTF_Salida )
      I_Contact( #DCARGARRA_ET01 )
   END_RUNG wire#w2
   RUNG wire#w1
      Contact( #HorqGarra_EnOperacion )
      Contact( #Interlock_Horquilla.RecogerCarga_SalidaHorq )
      wire#w3
      Coil( #Interlock_Garras.DejarCarga_EntradaGarra )
   END_RUNG
   RUNG wire#w1
      Contact( #Elev_DesCargaEnGarra )
      Contact( #DCARGARRA_ET03 )
   END_RUNG wire#w3
   // the same network as SCL:
   #Interlock_Garras.AVTF_EntradaGarra := "ON" AND ((#HorqGarra_EnOperacion AND #Interlock_Horquilla.AVTF_SalidaHorq) OR (#Elev_DesCargaEnGarra AND #Interlock_TELEV.AVTF_Salida AND NOT #DCARGARRA_ET01));
   #Interlock_Garras.DejarCarga_EntradaGarra := "ON" AND ((#HorqGarra_EnOperacion AND #Interlock_Horquilla.RecogerCarga_SalidaHorq) OR (#Elev_DesCargaEnGarra AND #DCARGARRA_ET03));
END_REGION

REGION Network 68: Interlock de Salida la Garra
   // Operacion --> De Garra al Elevador
   RUNG wire#powerrail
      Contact( "ON" )
      wire#w1
      Contact( #Elev_CargaDeGarra )
      Contact( #Interlock_TELEV.PTF_Entrada )
      Contact( #CheckElev_EnGarra )
      Coil( #Interlock_Garras.PTF_SalidaGarra )
   END_RUNG
   RUNG wire#w1
      Contact( #Elev_CargaDeGarra )
      Contact( #Interlock_TELEV.FTF_Entrada )
      Coil( #Interlock_Garras.FTF_SalidaGarra )
   END_RUNG
   RUNG wire#w1
      Contact( #Elev_CargaDeGarra )
      I_Contact( #CARGARRA_ET01 )
      I_Contact( #CARGARRA_ET05 )
      Contact( #CheckElev_EnGarra )
      Coil( #Interlock_Garras.OrdenDeSalida )
   END_RUNG
   RUNG wire#w1
      Contact( #Elev_CargaDeGarra )
      Contact( #CARGARRA_ET04 )
      Coil( #Interlock_Garras.RecogidaCarga_SalidaGarra )
   END_RUNG
   // the same network as SCL:
   #Interlock_Garras.PTF_SalidaGarra := "ON" AND #Elev_CargaDeGarra AND #Interlock_TELEV.PTF_Entrada AND #CheckElev_EnGarra;
   #Interlock_Garras.FTF_SalidaGarra := "ON" AND #Elev_CargaDeGarra AND #Interlock_TELEV.FTF_Entrada;
   #Interlock_Garras.OrdenDeSalida := "ON" AND #Elev_CargaDeGarra AND NOT #CARGARRA_ET01 AND NOT #CARGARRA_ET05 AND #CheckElev_EnGarra;
   #Interlock_Garras.RecogidaCarga_SalidaGarra := "ON" AND #Elev_CargaDeGarra AND #CARGARRA_ET04;
END_REGION

REGION Network 69: Interlock de Entrada a la Horquilla
   // Operacion --> Paleta  del Elevador a la Horquilla
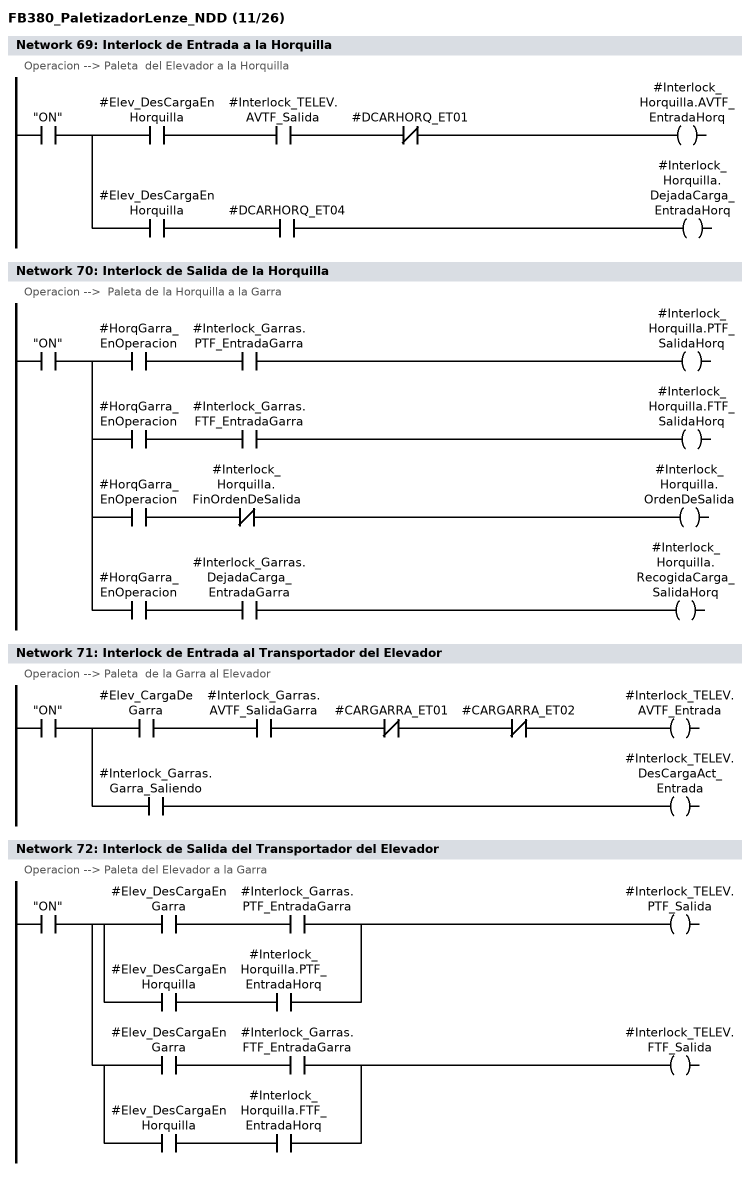
   RUNG wire#powerrail
      Contact( "ON" )
      wire#w1
      Contact( #Elev_DesCargaEnHorquilla )
      Contact( #Interlock_TELEV.AVTF_Salida )
      I_Contact( #DCARHORQ_ET01 )
      Coil( #Interlock_Horquilla.AVTF_EntradaHorq )
   END_RUNG
   RUNG wire#w1
      Contact( #Elev_DesCargaEnHorquilla )
      Contact( #DCARHORQ_ET04 )
      Coil( #Interlock_Horquilla.DejadaCarga_EntradaHorq )
   END_RUNG
   // the same network as SCL:
   #Interlock_Horquilla.AVTF_EntradaHorq := "ON" AND #Elev_DesCargaEnHorquilla AND #Interlock_TELEV.AVTF_Salida AND NOT #DCARHORQ_ET01;
   #Interlock_Horquilla.DejadaCarga_EntradaHorq := "ON" AND #Elev_DesCargaEnHorquilla AND #DCARHORQ_ET04;
END_REGION

REGION Network 70: Interlock de Salida de la Horquilla
   // Operacion -->  Paleta de la Horquilla a la Garra
   RUNG wire#powerrail
      Contact( "ON" )
      wire#w1
      Contact( #HorqGarra_EnOperacion )
      Contact( #Interlock_Garras.PTF_EntradaGarra )
      Coil( #Interlock_Horquilla.PTF_SalidaHorq )
   END_RUNG
   RUNG wire#w1
      Contact( #HorqGarra_EnOperacion )
      Contact( #Interlock_Garras.FTF_EntradaGarra )
      Coil( #Interlock_Horquilla.FTF_SalidaHorq )
   END_RUNG
   RUNG wire#w1
      Contact( #HorqGarra_EnOperacion )
      I_Contact( #Interlock_Horquilla.FinOrdenDeSalida )
      Coil( #Interlock_Horquilla.OrdenDeSalida )
   END_RUNG
   RUNG wire#w1
      Contact( #HorqGarra_EnOperacion )
      Contact( #Interlock_Garras.DejadaCarga_EntradaGarra )
      Coil( #Interlock_Horquilla.RecogidaCarga_SalidaHorq )
   END_RUNG
   // the same network as SCL:
   #Interlock_Horquilla.PTF_SalidaHorq := "ON" AND #HorqGarra_EnOperacion AND #Interlock_Garras.PTF_EntradaGarra;
   #Interlock_Horquilla.FTF_SalidaHorq := "ON" AND #HorqGarra_EnOperacion AND #Interlock_Garras.FTF_EntradaGarra;
   #Interlock_Horquilla.OrdenDeSalida := "ON" AND #HorqGarra_EnOperacion AND NOT #Interlock_Horquilla.FinOrdenDeSalida;
   #Interlock_Horquilla.RecogidaCarga_SalidaHorq := "ON" AND #HorqGarra_EnOperacion AND #Interlock_Garras.DejadaCarga_EntradaGarra;
END_REGION

REGION Network 71: Interlock de Entrada al Transportador del Elevador
   // Operacion --> Paleta  de la Garra al Elevador
   RUNG wire#powerrail
      Contact( "ON" )
      wire#w1
      Contact( #Elev_CargaDeGarra )
      Contact( #Interlock_Garras.AVTF_SalidaGarra )
      I_Contact( #CARGARRA_ET01 )
      I_Contact( #CARGARRA_ET02 )
      Coil( #Interlock_TELEV.AVTF_Entrada )
   END_RUNG
   RUNG wire#w1
      Contact( #Interlock_Garras.Garra_Saliendo )
      Coil( #Interlock_TELEV.DesCargaAct_Entrada )
   END_RUNG
   // the same network as SCL:
   #Interlock_TELEV.AVTF_Entrada := "ON" AND #Elev_CargaDeGarra AND #Interlock_Garras.AVTF_SalidaGarra AND NOT #CARGARRA_ET01 AND NOT #CARGARRA_ET02;
   #Interlock_TELEV.DesCargaAct_Entrada := "ON" AND #Interlock_Garras.Garra_Saliendo;
END_REGION

REGION Network 72: Interlock de Salida del Transportador del Elevador
   // Operacion --> Paleta del Elevador a la Garra
   RUNG wire#powerrail
      Contact( "ON" )
      wire#w1
      Contact( #Elev_DesCargaEnGarra )
      Contact( #Interlock_Garras.PTF_EntradaGarra )
      wire#w2
      Coil( #Interlock_TELEV.PTF_Salida )
   END_RUNG
   RUNG wire#w1
      Contact( #Elev_DesCargaEnHorquilla )
      Contact( #Interlock_Horquilla.PTF_EntradaHorq )
   END_RUNG wire#w2
   RUNG wire#w1
      Contact( #Elev_DesCargaEnGarra )
      Contact( #Interlock_Garras.FTF_EntradaGarra )
      wire#w3
      Coil( #Interlock_TELEV.FTF_Salida )
   END_RUNG
   RUNG wire#w1
      Contact( #Elev_DesCargaEnHorquilla )
      Contact( #Interlock_Horquilla.FTF_EntradaHorq )
   END_RUNG wire#w3
   // the same network as SCL:
   #Interlock_TELEV.PTF_Salida := "ON" AND ((#Elev_DesCargaEnGarra AND #Interlock_Garras.PTF_EntradaGarra) OR (#Elev_DesCargaEnHorquilla AND #Interlock_Horquilla.PTF_EntradaHorq));
   #Interlock_TELEV.FTF_Salida := "ON" AND ((#Elev_DesCargaEnGarra AND #Interlock_Garras.FTF_EntradaGarra) OR (#Elev_DesCargaEnHorquilla AND #Interlock_Horquilla.FTF_EntradaHorq));
END_REGION

REGION Network 73: ---
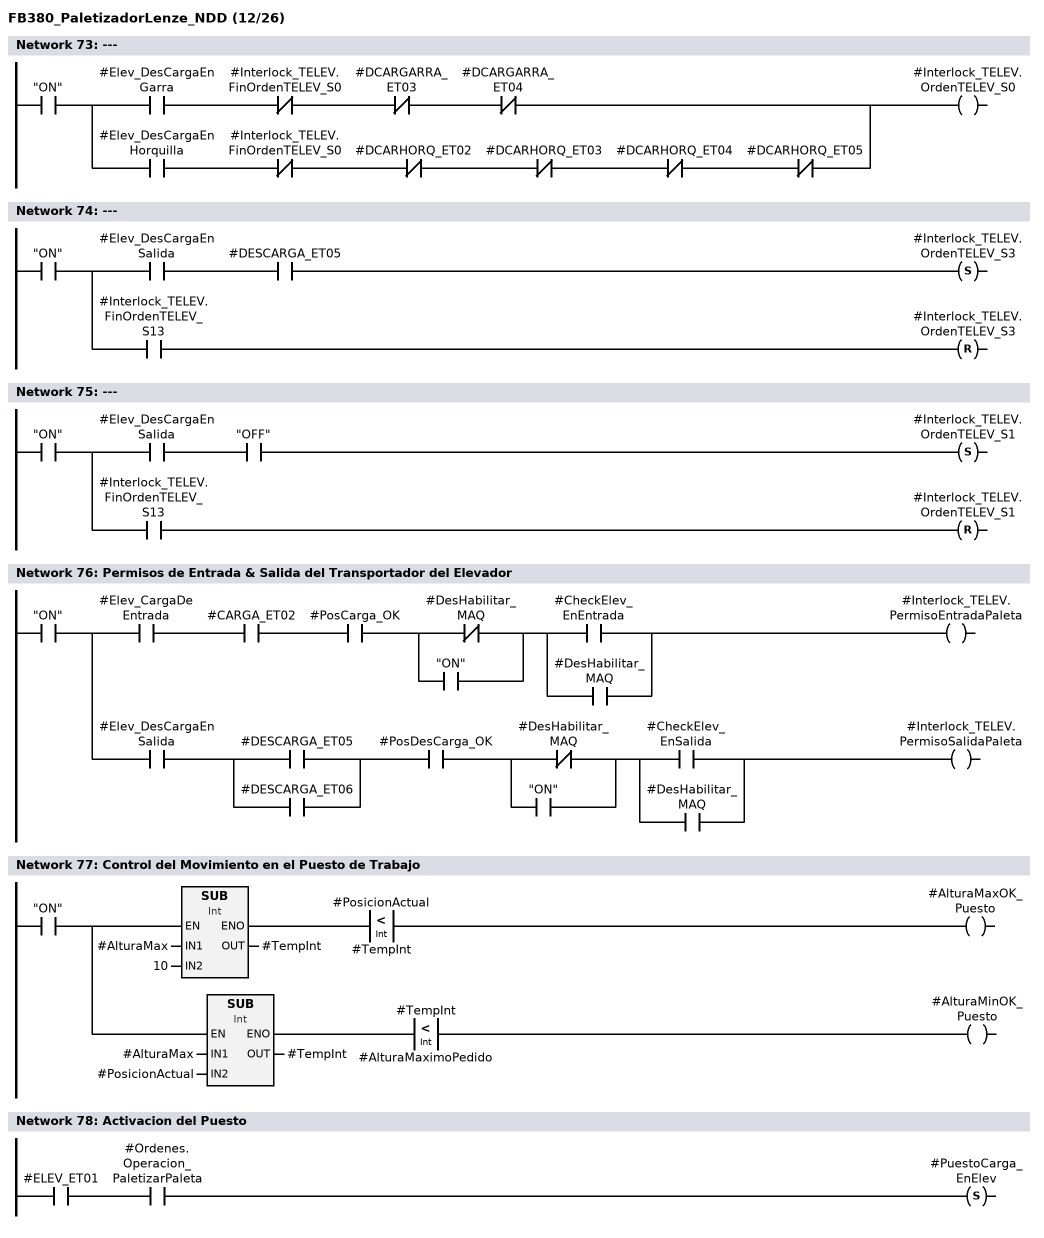
   RUNG wire#powerrail
      Contact( "ON" )
      wire#w1
      Contact( #Elev_DesCargaEnGarra )
      I_Contact( #Interlock_TELEV.FinOrdenTELEV_S0 )
      I_Contact( #DCARGARRA_ET03 )
      I_Contact( #DCARGARRA_ET04 )
      wire#w2
      Coil( #Interlock_TELEV.OrdenTELEV_S0 )
   END_RUNG
   RUNG wire#w1
      Contact( #Elev_DesCargaEnHorquilla )
      I_Contact( #Interlock_TELEV.FinOrdenTELEV_S0 )
      I_Contact( #DCARHORQ_ET02 )
      I_Contact( #DCARHORQ_ET03 )
      I_Contact( #DCARHORQ_ET04 )
      I_Contact( #DCARHORQ_ET05 )
   END_RUNG wire#w2
   // the same network as SCL:
   #Interlock_TELEV.OrdenTELEV_S0 := "ON" AND ((#Elev_DesCargaEnGarra AND NOT #Interlock_TELEV.FinOrdenTELEV_S0 AND NOT #DCARGARRA_ET03 AND NOT #DCARGARRA_ET04) OR (#Elev_DesCargaEnHorquilla AND NOT #Interlock_TELEV.FinOrdenTELEV_S0 AND NOT #DCARHORQ_ET02 AND NOT #DCARHORQ_ET03 AND NOT #DCARHORQ_ET04 AND NOT #DCARHORQ_ET05));
END_REGION

REGION Network 74: ---
   RUNG wire#powerrail
      Contact( "ON" )
      wire#w1
      Contact( #Elev_DesCargaEnSalida )
      Contact( #DESCARGA_ET05 )
      S_Coil( #Interlock_TELEV.OrdenTELEV_S3 )
   END_RUNG
   RUNG wire#w1
      Contact( #Interlock_TELEV.FinOrdenTELEV_S13 )
      R_Coil( #Interlock_TELEV.OrdenTELEV_S3 )
   END_RUNG
   // the same network as SCL:
   IF "ON" AND #Elev_DesCargaEnSalida AND #DESCARGA_ET05 THEN #Interlock_TELEV.OrdenTELEV_S3 := TRUE; END_IF;
   IF "ON" AND #Interlock_TELEV.FinOrdenTELEV_S13 THEN #Interlock_TELEV.OrdenTELEV_S3 := FALSE; END_IF;
END_REGION

REGION Network 75: ---
   RUNG wire#powerrail
      Contact( "ON" )
      wire#w1
      Contact( #Elev_DesCargaEnSalida )
      Contact( "OFF" )
      S_Coil( #Interlock_TELEV.OrdenTELEV_S1 )
   END_RUNG
   RUNG wire#w1
      Contact( #Interlock_TELEV.FinOrdenTELEV_S13 )
      R_Coil( #Interlock_TELEV.OrdenTELEV_S1 )
   END_RUNG
   // the same network as SCL:
   IF "ON" AND #Elev_DesCargaEnSalida AND "OFF" THEN #Interlock_TELEV.OrdenTELEV_S1 := TRUE; END_IF;
   IF "ON" AND #Interlock_TELEV.FinOrdenTELEV_S13 THEN #Interlock_TELEV.OrdenTELEV_S1 := FALSE; END_IF;
END_REGION

REGION Network 76: Permisos de Entrada & Salida del Transportador del Elevador
   RUNG wire#powerrail
      Contact( "ON" )
      wire#w1
      Contact( #Elev_CargaDeEntrada )
      Contact( #CARGA_ET02 )
      Contact( #PosCarga_OK )
      wire#w2
      I_Contact( #DesHabilitar_MAQ )
      wire#w3
      Contact( #CheckElev_EnEntrada )
      wire#w4
      Coil( #Interlock_TELEV.PermisoEntradaPaleta )
   END_RUNG
   RUNG wire#w2
      Contact( "ON" )
   END_RUNG wire#w3
   RUNG wire#w3
      Contact( #DesHabilitar_MAQ )
   END_RUNG wire#w4
   RUNG wire#w1
      Contact( #Elev_DesCargaEnSalida )
      wire#w5
      Contact( #DESCARGA_ET05 )
      wire#w6
      Contact( #PosDesCarga_OK )
      wire#w7
      I_Contact( #DesHabilitar_MAQ )
      wire#w8
      Contact( #CheckElev_EnSalida )
      wire#w9
      Coil( #Interlock_TELEV.PermisoSalidaPaleta )
   END_RUNG
   RUNG wire#w5
      Contact( #DESCARGA_ET06 )
   END_RUNG wire#w6
   RUNG wire#w7
      Contact( "ON" )
   END_RUNG wire#w8
   RUNG wire#w8
      Contact( #DesHabilitar_MAQ )
   END_RUNG wire#w9
   // the same network as SCL:
   #Interlock_TELEV.PermisoEntradaPaleta := "ON" AND #Elev_CargaDeEntrada AND #CARGA_ET02 AND #PosCarga_OK AND (NOT #DesHabilitar_MAQ OR "ON") AND (#CheckElev_EnEntrada OR #DesHabilitar_MAQ);
   #Interlock_TELEV.PermisoSalidaPaleta := "ON" AND #Elev_DesCargaEnSalida AND (#DESCARGA_ET05 OR #DESCARGA_ET06) AND #PosDesCarga_OK AND (NOT #DesHabilitar_MAQ OR "ON") AND (#CheckElev_EnSalida OR #DesHabilitar_MAQ);
END_REGION

REGION Network 77: Control del Movimiento en el Puesto de Trabajo
   RUNG wire#powerrail
      Contact( "ON" )
      wire#w1
      { S7_Templates := "SrcType := Int"; S7_GenerateENO := "TRUE" } Sub(in1 := #AlturaMax, in2 := 10, out => #TempInt)
      { S7_Templates := "SrcType := Int" } LT_Contact(in1 := #PosicionActual, in2 := #TempInt)
      Coil( #AlturaMaxOK_Puesto )
   END_RUNG
   RUNG wire#w1
      { S7_Templates := "SrcType := Int"; S7_GenerateENO := "TRUE" } Sub(in1 := #AlturaMax, in2 := #PosicionActual, out => #TempInt)
      { S7_Templates := "SrcType := Int" } LT_Contact(in1 := #TempInt, in2 := #AlturaMaximoPedido)
      Coil( #AlturaMinOK_Puesto )
   END_RUNG
   // the same network as SCL:
   // ENO of a box is taken as its EN; it also drops when the box reports an error
   IF "ON" THEN #TempInt := #AlturaMax - 10; END_IF;
   #AlturaMaxOK_Puesto := "ON" AND (#PosicionActual < #TempInt);
   IF "ON" THEN #TempInt := #AlturaMax - #PosicionActual; END_IF;
   #AlturaMinOK_Puesto := "ON" AND (#TempInt < #AlturaMaximoPedido);
END_REGION

REGION Network 78: Activacion del Puesto
   RUNG wire#powerrail
      Contact( #ELEV_ET01 )
      Contact( #Ordenes.Operacion_PaletizarPaleta )
      S_Coil( #PuestoCarga_EnElev )
   END_RUNG
   // the same network as SCL:
   IF #ELEV_ET01 AND #Ordenes.Operacion_PaletizarPaleta THEN #PuestoCarga_EnElev := TRUE; END_IF;
END_REGION

REGION Network 79: ---
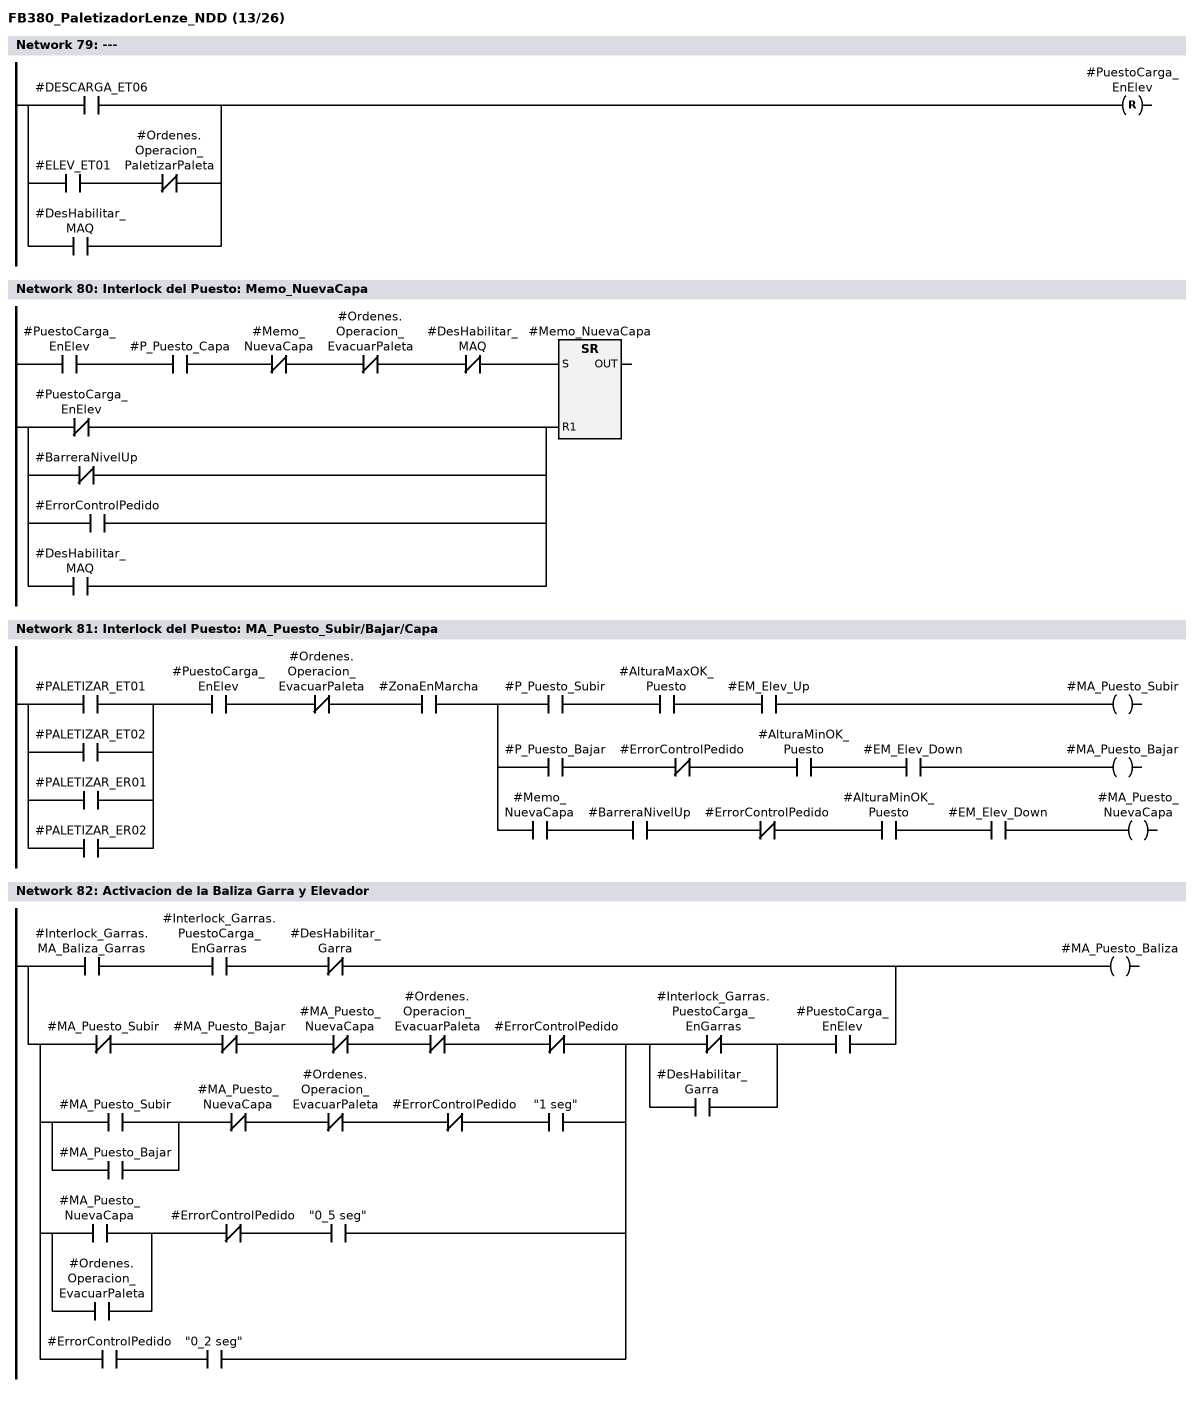
   RUNG wire#powerrail
      Contact( #DESCARGA_ET06 )
      wire#w1
      R_Coil( #PuestoCarga_EnElev )
   END_RUNG
   RUNG wire#powerrail
      Contact( #ELEV_ET01 )
      I_Contact( #Ordenes.Operacion_PaletizarPaleta )
   END_RUNG wire#w1
   RUNG wire#powerrail
      Contact( #DesHabilitar_MAQ )
   END_RUNG wire#w1
   // the same network as SCL:
   IF #DESCARGA_ET06 OR (#ELEV_ET01 AND NOT #Ordenes.Operacion_PaletizarPaleta) OR #DesHabilitar_MAQ THEN
       #PuestoCarga_EnElev := FALSE;
   END_IF;
END_REGION

REGION Network 80: Interlock del Puesto: Memo_NuevaCapa
   RUNG wire#powerrail
      Contact( #PuestoCarga_EnElev )
      Contact( #P_Puesto_Capa )
      I_Contact( #Memo_NuevaCapa )
      I_Contact( #Ordenes.Operacion_EvacuarPaleta )
      I_Contact( #DesHabilitar_MAQ )
      S_SR(operand := #Memo_NuevaCapa, r1 := wire#w1)
   END_RUNG
   RUNG wire#powerrail
      I_Contact( #PuestoCarga_EnElev )
   END_RUNG wire#w1
   RUNG wire#powerrail
      I_Contact( #BarreraNivelUp )
   END_RUNG wire#w1
   RUNG wire#powerrail
      Contact( #ErrorControlPedido )
   END_RUNG wire#w1
   RUNG wire#powerrail
      Contact( #DesHabilitar_MAQ )
   END_RUNG wire#w1
   // the same network as SCL:
   IF #PuestoCarga_EnElev AND #P_Puesto_Capa AND NOT #Memo_NuevaCapa AND NOT #Ordenes.Operacion_EvacuarPaleta AND NOT #DesHabilitar_MAQ THEN
       #Memo_NuevaCapa := TRUE;   // SR flip-flop
   END_IF;
   IF NOT #PuestoCarga_EnElev OR NOT #BarreraNivelUp OR #ErrorControlPedido OR #DesHabilitar_MAQ THEN
       #Memo_NuevaCapa := FALSE;
   END_IF;
END_REGION

REGION Network 81: Interlock del Puesto: MA_Puesto_Subir/Bajar/Capa
   RUNG wire#powerrail
      Contact( #PALETIZAR_ET01 )
      wire#w1
      Contact( #PuestoCarga_EnElev )
      I_Contact( #Ordenes.Operacion_EvacuarPaleta )
      Contact( #ZonaEnMarcha )
      wire#w2
      Contact( #P_Puesto_Subir )
      Contact( #AlturaMaxOK_Puesto )
      Contact( #EM_Elev_Up )
      Coil( #MA_Puesto_Subir )
   END_RUNG
   RUNG wire#powerrail
      Contact( #PALETIZAR_ET02 )
   END_RUNG wire#w1
   RUNG wire#powerrail
      Contact( #PALETIZAR_ER01 )
   END_RUNG wire#w1
   RUNG wire#powerrail
      Contact( #PALETIZAR_ER02 )
   END_RUNG wire#w1
   RUNG wire#w2
      Contact( #P_Puesto_Bajar )
      I_Contact( #ErrorControlPedido )
      Contact( #AlturaMinOK_Puesto )
      Contact( #EM_Elev_Down )
      Coil( #MA_Puesto_Bajar )
   END_RUNG
   RUNG wire#w2
      Contact( #Memo_NuevaCapa )
      Contact( #BarreraNivelUp )
      I_Contact( #ErrorControlPedido )
      Contact( #AlturaMinOK_Puesto )
      Contact( #EM_Elev_Down )
      Coil( #MA_Puesto_NuevaCapa )
   END_RUNG
   // the same network as SCL:
   #_w1 := (#PALETIZAR_ET01 OR #PALETIZAR_ET02 OR #PALETIZAR_ER01 OR #PALETIZAR_ER02) AND #PuestoCarga_EnElev AND NOT #Ordenes.Operacion_EvacuarPaleta AND #ZonaEnMarcha;
   #MA_Puesto_Subir := #_w1 AND #P_Puesto_Subir AND #AlturaMaxOK_Puesto AND #EM_Elev_Up;
   #MA_Puesto_Bajar := #_w1 AND #P_Puesto_Bajar AND NOT #ErrorControlPedido AND #AlturaMinOK_Puesto AND #EM_Elev_Down;
   #MA_Puesto_NuevaCapa := #_w1 AND #Memo_NuevaCapa AND #BarreraNivelUp AND NOT #ErrorControlPedido AND #AlturaMinOK_Puesto AND #EM_Elev_Down;
END_REGION

REGION Network 82: Activacion de la Baliza Garra y Elevador
   RUNG wire#powerrail
      Contact( #Interlock_Garras.MA_Baliza_Garras )
      Contact( #Interlock_Garras.PuestoCarga_EnGarras )
      I_Contact( #DesHabilitar_Garra )
      wire#w1
      Coil( #MA_Puesto_Baliza )
   END_RUNG
   RUNG wire#powerrail
      I_Contact( #MA_Puesto_Subir )
      I_Contact( #MA_Puesto_Bajar )
      I_Contact( #MA_Puesto_NuevaCapa )
      I_Contact( #Ordenes.Operacion_EvacuarPaleta )
      I_Contact( #ErrorControlPedido )
      wire#w2
      I_Contact( #Interlock_Garras.PuestoCarga_EnGarras )
      wire#w5
      Contact( #PuestoCarga_EnElev )
   END_RUNG wire#w1
   RUNG wire#powerrail
      Contact( #MA_Puesto_Subir )
      wire#w3
      I_Contact( #MA_Puesto_NuevaCapa )
      I_Contact( #Ordenes.Operacion_EvacuarPaleta )
      I_Contact( #ErrorControlPedido )
      Contact( "1 seg" )
   END_RUNG wire#w2
   RUNG wire#powerrail
      Contact( #MA_Puesto_Bajar )
   END_RUNG wire#w3
   RUNG wire#powerrail
      Contact( #MA_Puesto_NuevaCapa )
      wire#w4
      I_Contact( #ErrorControlPedido )
      Contact( "0_5 seg" )
   END_RUNG wire#w2
   RUNG wire#powerrail
      Contact( #Ordenes.Operacion_EvacuarPaleta )
   END_RUNG wire#w4
   RUNG wire#powerrail
      Contact( #ErrorControlPedido )
      Contact( "0_2 seg" )
   END_RUNG wire#w2
   RUNG wire#w2
      Contact( #DesHabilitar_Garra )
   END_RUNG wire#w5
   // the same network as SCL:
   #MA_Puesto_Baliza := (#Interlock_Garras.MA_Baliza_Garras AND #Interlock_Garras.PuestoCarga_EnGarras AND NOT #DesHabilitar_Garra) OR (((NOT #MA_Puesto_Subir AND NOT #MA_Puesto_Bajar AND NOT #MA_Puesto_NuevaCapa AND NOT #Ordenes.Operacion_EvacuarPaleta AND NOT #ErrorControlPedido) OR ((#MA_Puesto_Subir OR #MA_Puesto_Bajar) AND NOT #MA_Puesto_NuevaCapa AND NOT #Ordenes.Operacion_EvacuarPaleta AND NOT #ErrorControlPedido AND "1 seg") OR ((#MA_Puesto_NuevaCapa OR #Ordenes.Operacion_EvacuarPaleta) AND NOT #ErrorControlPedido AND "0_5 seg") OR (#ErrorControlPedido AND "0_2 seg")) AND (NOT #Interlock_Garras.PuestoCarga_EnGarras OR #DesHabilitar_Garra) AND #PuestoCarga_EnElev);
END_REGION

REGION Network 83: Control de Elevador - Ordenes
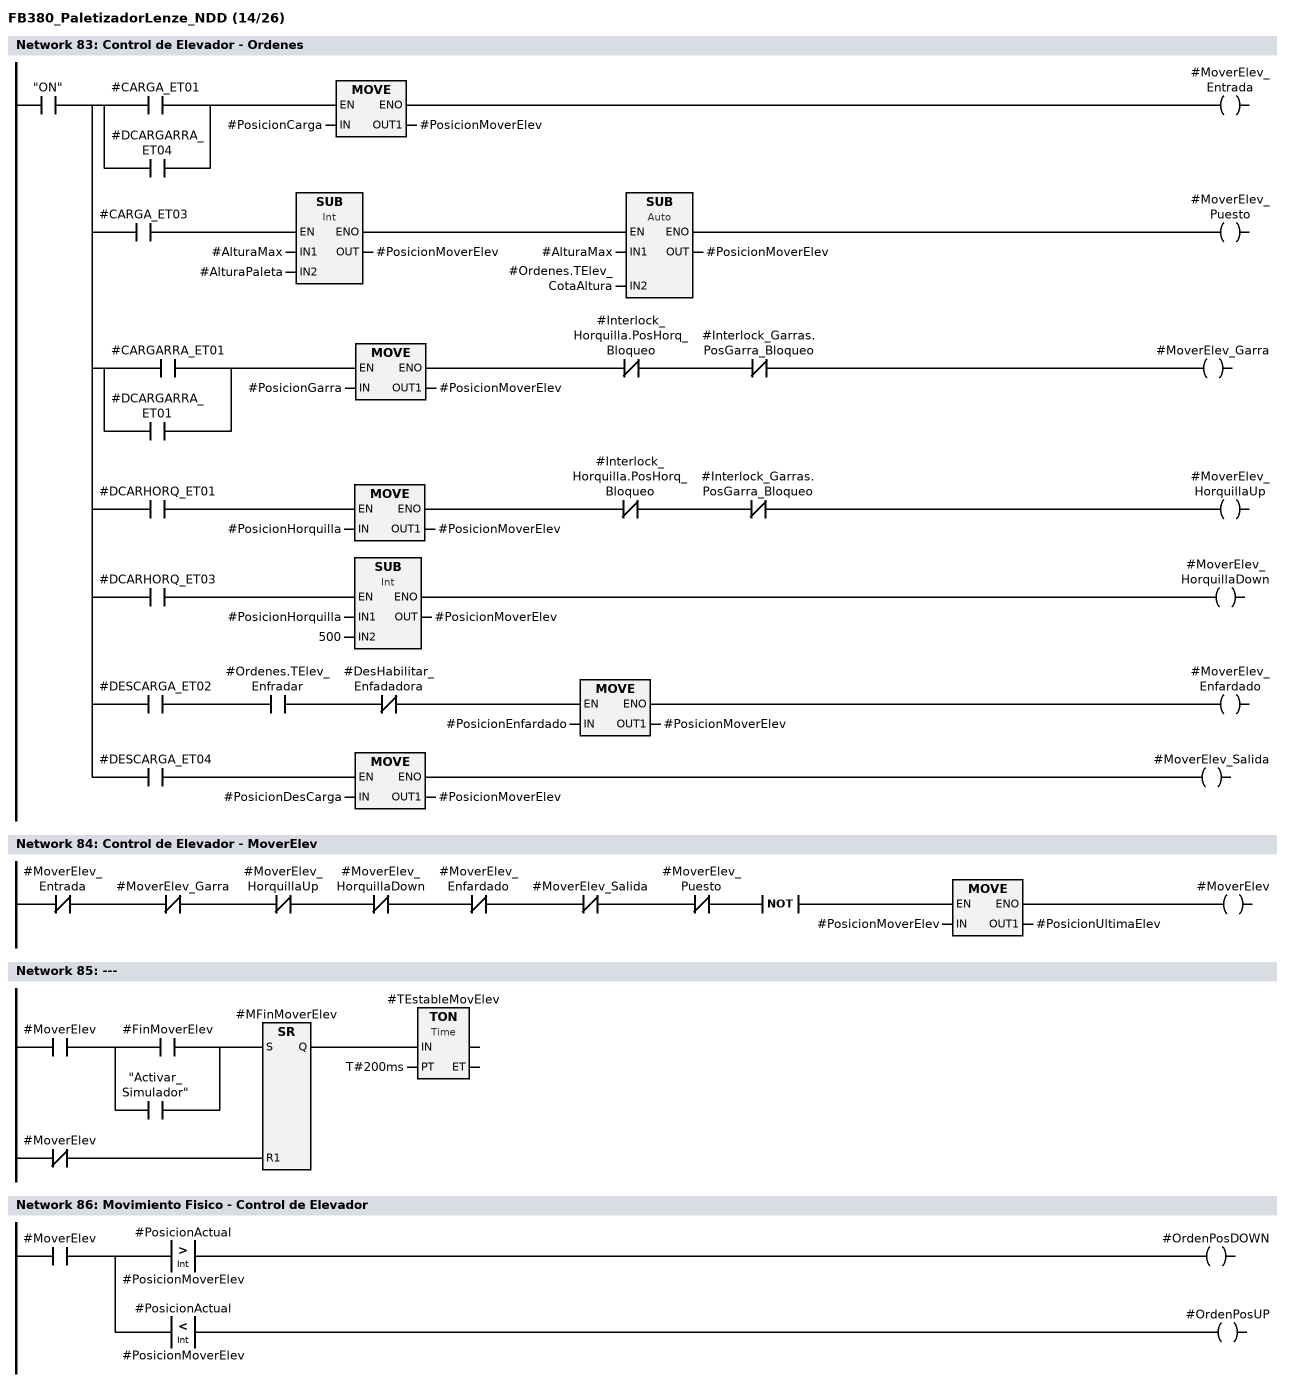
   RUNG wire#powerrail
      Contact( "ON" )
      wire#w1
      Contact( #CARGA_ET01 )
      wire#w2
      { S7_GenerateENO := "TRUE" } Move(in := #PosicionCarga, out1 => #PosicionMoverElev)
      Coil( #MoverElev_Entrada )
   END_RUNG
   RUNG wire#w1
      Contact( #DCARGARRA_ET04 )
   END_RUNG wire#w2
   RUNG wire#w1
      Contact( #CARGA_ET03 )
      { S7_Templates := "SrcType := Int"; S7_GenerateENO := "TRUE" } Sub(in1 := #AlturaMax, in2 := #AlturaPaleta, out => #PosicionMoverElev)
      Sub(in1 := #AlturaMax, in2 := #Ordenes.TElev_CotaAltura, out => #PosicionMoverElev)
      Coil( #MoverElev_Puesto )
   END_RUNG
   RUNG wire#w1
      Contact( #CARGARRA_ET01 )
      wire#w3
      { S7_GenerateENO := "TRUE" } Move(in := #PosicionGarra, out1 => #PosicionMoverElev)
      I_Contact( #Interlock_Horquilla.PosHorq_Bloqueo )
      I_Contact( #Interlock_Garras.PosGarra_Bloqueo )
      Coil( #MoverElev_Garra )
   END_RUNG
   RUNG wire#w1
      Contact( #DCARGARRA_ET01 )
   END_RUNG wire#w3
   RUNG wire#w1
      Contact( #DCARHORQ_ET01 )
      { S7_GenerateENO := "TRUE" } Move(in := #PosicionHorquilla, out1 => #PosicionMoverElev)
      I_Contact( #Interlock_Horquilla.PosHorq_Bloqueo )
      I_Contact( #Interlock_Garras.PosGarra_Bloqueo )
      Coil( #MoverElev_HorquillaUp )
   END_RUNG
   RUNG wire#w1
      Contact( #DCARHORQ_ET03 )
      { S7_Templates := "SrcType := Int"; S7_GenerateENO := "TRUE" } Sub(in1 := #PosicionHorquilla, in2 := 500, out => #PosicionMoverElev)
      Coil( #MoverElev_HorquillaDown )
   END_RUNG
   RUNG wire#w1
      Contact( #DESCARGA_ET02 )
      Contact( #Ordenes.TElev_Enfradar )
      I_Contact( #DesHabilitar_Enfadadora )
      { S7_GenerateENO := "TRUE" } Move(in := #PosicionEnfardado, out1 => #PosicionMoverElev)
      Coil( #MoverElev_Enfardado )
   END_RUNG
   RUNG wire#w1
      Contact( #DESCARGA_ET04 )
      { S7_GenerateENO := "TRUE" } Move(in := #PosicionDesCarga, out1 => #PosicionMoverElev)
      Coil( #MoverElev_Salida )
   END_RUNG
   // the same network as SCL:
   // ENO of a box is taken as its EN; it also drops when the box reports an error
   #_w1 := "ON" AND (#CARGA_ET01 OR #DCARGARRA_ET04);
   IF #_w1 THEN #PosicionMoverElev := #PosicionCarga; END_IF;
   #MoverElev_Entrada := #_w1;
   #_w2 := "ON" AND #CARGA_ET03;
   IF #_w2 THEN
       #PosicionMoverElev := #AlturaMax - #AlturaPaleta;
       #PosicionMoverElev := #AlturaMax - #Ordenes.TElev_CotaAltura;
   END_IF;
   #MoverElev_Puesto := #_w2;
   #_w3 := "ON" AND (#CARGARRA_ET01 OR #DCARGARRA_ET01);
   IF #_w3 THEN #PosicionMoverElev := #PosicionGarra; END_IF;
   #MoverElev_Garra := #_w3 AND NOT #Interlock_Horquilla.PosHorq_Bloqueo AND NOT #Interlock_Garras.PosGarra_Bloqueo;
   #_w4 := "ON" AND #DCARHORQ_ET01;
   IF #_w4 THEN #PosicionMoverElev := #PosicionHorquilla; END_IF;
   #MoverElev_HorquillaUp := #_w4 AND NOT #Interlock_Horquilla.PosHorq_Bloqueo AND NOT #Interlock_Garras.PosGarra_Bloqueo;
   #_w5 := "ON" AND #DCARHORQ_ET03;
   IF #_w5 THEN #PosicionMoverElev := #PosicionHorquilla - 500; END_IF;
   #MoverElev_HorquillaDown := #_w5;
   #_w6 := "ON" AND #DESCARGA_ET02 AND #Ordenes.TElev_Enfradar AND NOT #DesHabilitar_Enfadadora;
   IF #_w6 THEN #PosicionMoverElev := #PosicionEnfardado; END_IF;
   #MoverElev_Enfardado := #_w6;
   #_w7 := "ON" AND #DESCARGA_ET04;
   IF #_w7 THEN #PosicionMoverElev := #PosicionDesCarga; END_IF;
   #MoverElev_Salida := #_w7;
END_REGION

REGION Network 84: Control de Elevador - MoverElev
   RUNG wire#powerrail
      I_Contact( #MoverElev_Entrada )
      I_Contact( #MoverElev_Garra )
      I_Contact( #MoverElev_HorquillaUp )
      I_Contact( #MoverElev_HorquillaDown )
      I_Contact( #MoverElev_Enfardado )
      I_Contact( #MoverElev_Salida )
      I_Contact( #MoverElev_Puesto )
      Not()
      { S7_GenerateENO := "TRUE" } Move(in := #PosicionMoverElev, out1 => #PosicionUltimaElev)
      Coil( #MoverElev )
   END_RUNG
   // the same network as SCL:
   // ENO of a box is taken as its EN; it also drops when the box reports an error
   #_w1 := NOT (NOT #MoverElev_Entrada AND NOT #MoverElev_Garra AND NOT #MoverElev_HorquillaUp AND NOT #MoverElev_HorquillaDown AND NOT #MoverElev_Enfardado AND NOT #MoverElev_Salida AND NOT #MoverElev_Puesto);
   IF #_w1 THEN #PosicionUltimaElev := #PosicionMoverElev; END_IF;
   #MoverElev := #_w1;
END_REGION

REGION Network 85: ---
   RUNG wire#powerrail
      Contact( #MoverElev )
      wire#w1
      Contact( #FinMoverElev )
      wire#w2
      S_SR(operand := #MFinMoverElev, r1 := wire#w3)
      { S7_Templates := "time_type := Time" } #TEstableMovElev.TON(pt := T#200ms, et =>)
   END_RUNG
   RUNG wire#w1
      Contact( "Activar_Simulador" )
   END_RUNG wire#w2
   RUNG wire#powerrail
      I_Contact( #MoverElev )
   END_RUNG wire#w3
   // the same network as SCL:
   IF #MoverElev AND (#FinMoverElev OR "Activar_Simulador") THEN
       #MFinMoverElev := TRUE;   // SR flip-flop
   END_IF;
   IF NOT #MoverElev THEN #MFinMoverElev := FALSE; END_IF;
   #TEstableMovElev(IN := #MFinMoverElev, PT := T#200ms);   // TON
END_REGION

REGION Network 86: Movimiento Fisico - Control de Elevador
   RUNG wire#powerrail
      Contact( #MoverElev )
      wire#w1
      { S7_Templates := "SrcType := Int" } GT_Contact(in1 := #PosicionActual, in2 := #PosicionMoverElev)
      Coil( #OrdenPosDOWN )
   END_RUNG
   RUNG wire#w1
      { S7_Templates := "SrcType := Int" } LT_Contact(in1 := #PosicionActual, in2 := #PosicionMoverElev)
      Coil( #OrdenPosUP )
   END_RUNG
   // the same network as SCL:
   #OrdenPosDOWN := #MoverElev AND (#PosicionActual > #PosicionMoverElev);
   #OrdenPosUP := #MoverElev AND (#PosicionActual < #PosicionMoverElev);
END_REGION

REGION Network 87: ---
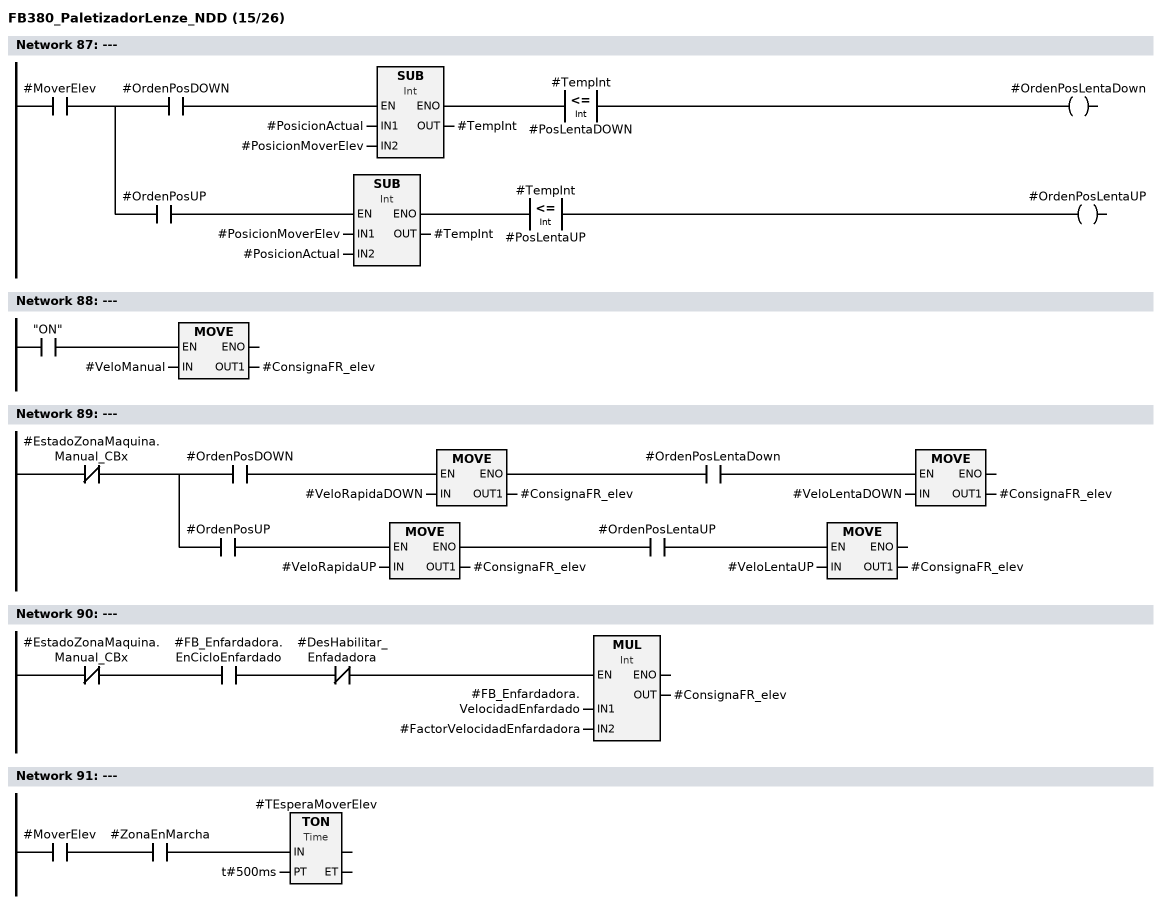
   RUNG wire#powerrail
      Contact( #MoverElev )
      wire#w1
      Contact( #OrdenPosDOWN )
      { S7_Templates := "SrcType := Int"; S7_GenerateENO := "TRUE" } Sub(in1 := #PosicionActual, in2 := #PosicionMoverElev, out => #TempInt)
      { S7_Templates := "SrcType := Int" } LE_Contact(in1 := #TempInt, in2 := #PosLentaDOWN)
      Coil( #OrdenPosLentaDown )
   END_RUNG
   RUNG wire#w1
      Contact( #OrdenPosUP )
      { S7_Templates := "SrcType := Int"; S7_GenerateENO := "TRUE" } Sub(in1 := #PosicionMoverElev, in2 := #PosicionActual, out => #TempInt)
      { S7_Templates := "SrcType := Int" } LE_Contact(in1 := #TempInt, in2 := #PosLentaUP)
      Coil( #OrdenPosLentaUP )
   END_RUNG
   // the same network as SCL:
   // ENO of a box is taken as its EN; it also drops when the box reports an error
   #_w1 := #MoverElev AND #OrdenPosDOWN;
   IF #_w1 THEN #TempInt := #PosicionActual - #PosicionMoverElev; END_IF;
   #OrdenPosLentaDown := #_w1 AND (#TempInt <= #PosLentaDOWN);
   #_w2 := #MoverElev AND #OrdenPosUP;
   IF #_w2 THEN #TempInt := #PosicionMoverElev - #PosicionActual; END_IF;
   #OrdenPosLentaUP := #_w2 AND (#TempInt <= #PosLentaUP);
END_REGION

REGION Network 88: ---
   RUNG wire#powerrail
      Contact( "ON" )
      { S7_GenerateENO := "TRUE" } Move(in := #VeloManual, out1 => #ConsignaFR_elev)
   END_RUNG
   // the same network as SCL:
   IF "ON" THEN #ConsignaFR_elev := #VeloManual; END_IF;
END_REGION

REGION Network 89: ---
   RUNG wire#powerrail
      I_Contact( #EstadoZonaMaquina.Manual_CBx )
      wire#w1
      Contact( #OrdenPosDOWN )
      { S7_GenerateENO := "TRUE" } Move(in := #VeloRapidaDOWN, out1 => #ConsignaFR_elev)
      Contact( #OrdenPosLentaDown )
      { S7_GenerateENO := "TRUE" } Move(in := #VeloLentaDOWN, out1 => #ConsignaFR_elev)
   END_RUNG
   RUNG wire#w1
      Contact( #OrdenPosUP )
      { S7_GenerateENO := "TRUE" } Move(in := #VeloRapidaUP, out1 => #ConsignaFR_elev)
      Contact( #OrdenPosLentaUP )
      { S7_GenerateENO := "TRUE" } Move(in := #VeloLentaUP, out1 => #ConsignaFR_elev)
   END_RUNG
   // the same network as SCL:
   // ENO of a box is taken as its EN; it also drops when the box reports an error
   #_w1 := NOT #EstadoZonaMaquina.Manual_CBx;
   #_w2 := #_w1 AND #OrdenPosDOWN;
   IF #_w2 THEN #ConsignaFR_elev := #VeloRapidaDOWN; END_IF;
   IF #_w2 AND #OrdenPosLentaDown THEN #ConsignaFR_elev := #VeloLentaDOWN; END_IF;
   #_w3 := #_w1 AND #OrdenPosUP;
   IF #_w3 THEN #ConsignaFR_elev := #VeloRapidaUP; END_IF;
   IF #_w3 AND #OrdenPosLentaUP THEN #ConsignaFR_elev := #VeloLentaUP; END_IF;
END_REGION

REGION Network 90: ---
   RUNG wire#powerrail
      I_Contact( #EstadoZonaMaquina.Manual_CBx )
      Contact( #FB_Enfardadora.EnCicloEnfardado )
      I_Contact( #DesHabilitar_Enfadadora )
      { S7_Templates := "SrcType := Int"; S7_GenerateENO := "TRUE" } Mul(in1 := #FB_Enfardadora.VelocidadEnfardado, in2 := #FactorVelocidadEnfardadora, out => #ConsignaFR_elev)
   END_RUNG
   // the same network as SCL:
   IF NOT #EstadoZonaMaquina.Manual_CBx AND #FB_Enfardadora.EnCicloEnfardado AND NOT #DesHabilitar_Enfadadora THEN
       #ConsignaFR_elev := #FB_Enfardadora.VelocidadEnfardado * #FactorVelocidadEnfardadora;
   END_IF;
END_REGION

REGION Network 91: ---
   RUNG wire#powerrail
      Contact( #MoverElev )
      Contact( #ZonaEnMarcha )
      { S7_Templates := "time_type := Time" } #TEsperaMoverElev.TON(pt := t#500ms, et =>)
   END_RUNG
   // the same network as SCL:
   #TEsperaMoverElev(IN := #MoverElev AND #ZonaEnMarcha, PT := t#500ms);   // TON
END_REGION

NETWORK
TITLE = ---
/////////////////////////////////////////////////////////////////////////
// Estado para el Movimiento de Elevacion

      L     P##EstadoZonaMovElev;  // Puntero a Estado ZONA
      T     #P_EstadoZonaMovElev;

      L     0;  // Inicilizo
      T     LW [#P_EstadoZonaMovElev];

// Automatico - Manual

      A     #EstadoZonaMesa.Automatico_CBx;
      =     #EstadoZonaMovElev.Automatico_CBx;

      A     #EstadoZonaMesa.Manual_CBx;
      =     #EstadoZonaMovElev.Manual_CBx;

// Marcha - Paro - Error

      A     #EstadoZonaMesa.Marcha_CBx;
      =     #EstadoZonaMovElev.Marcha_CBx;

      A     #EstadoZonaMesa.Paro_CBx;
      =     #EstadoZonaMovElev.Paro_CBx;

      A     #EstadoZonaMesa.Error_CBx;
      O     #EstadoZonaMaquina.Error_CBx;
      =     #EstadoZonaMovElev.Error_CBx;

// Reset

      A     #EstadoZonaMesa.Resetear_CBx;
      =     #EstadoZonaMovElev.Resetear_CBx;

// Rearme

      A     #EstadoZonaMesa.Rearme_CBx;
      O     #EstadoZonaMaquina.Rearme_CBx;
      =     #EstadoZonaMovElev.Rearme_CBx;



REGION Network 93: Control de la Elevacion
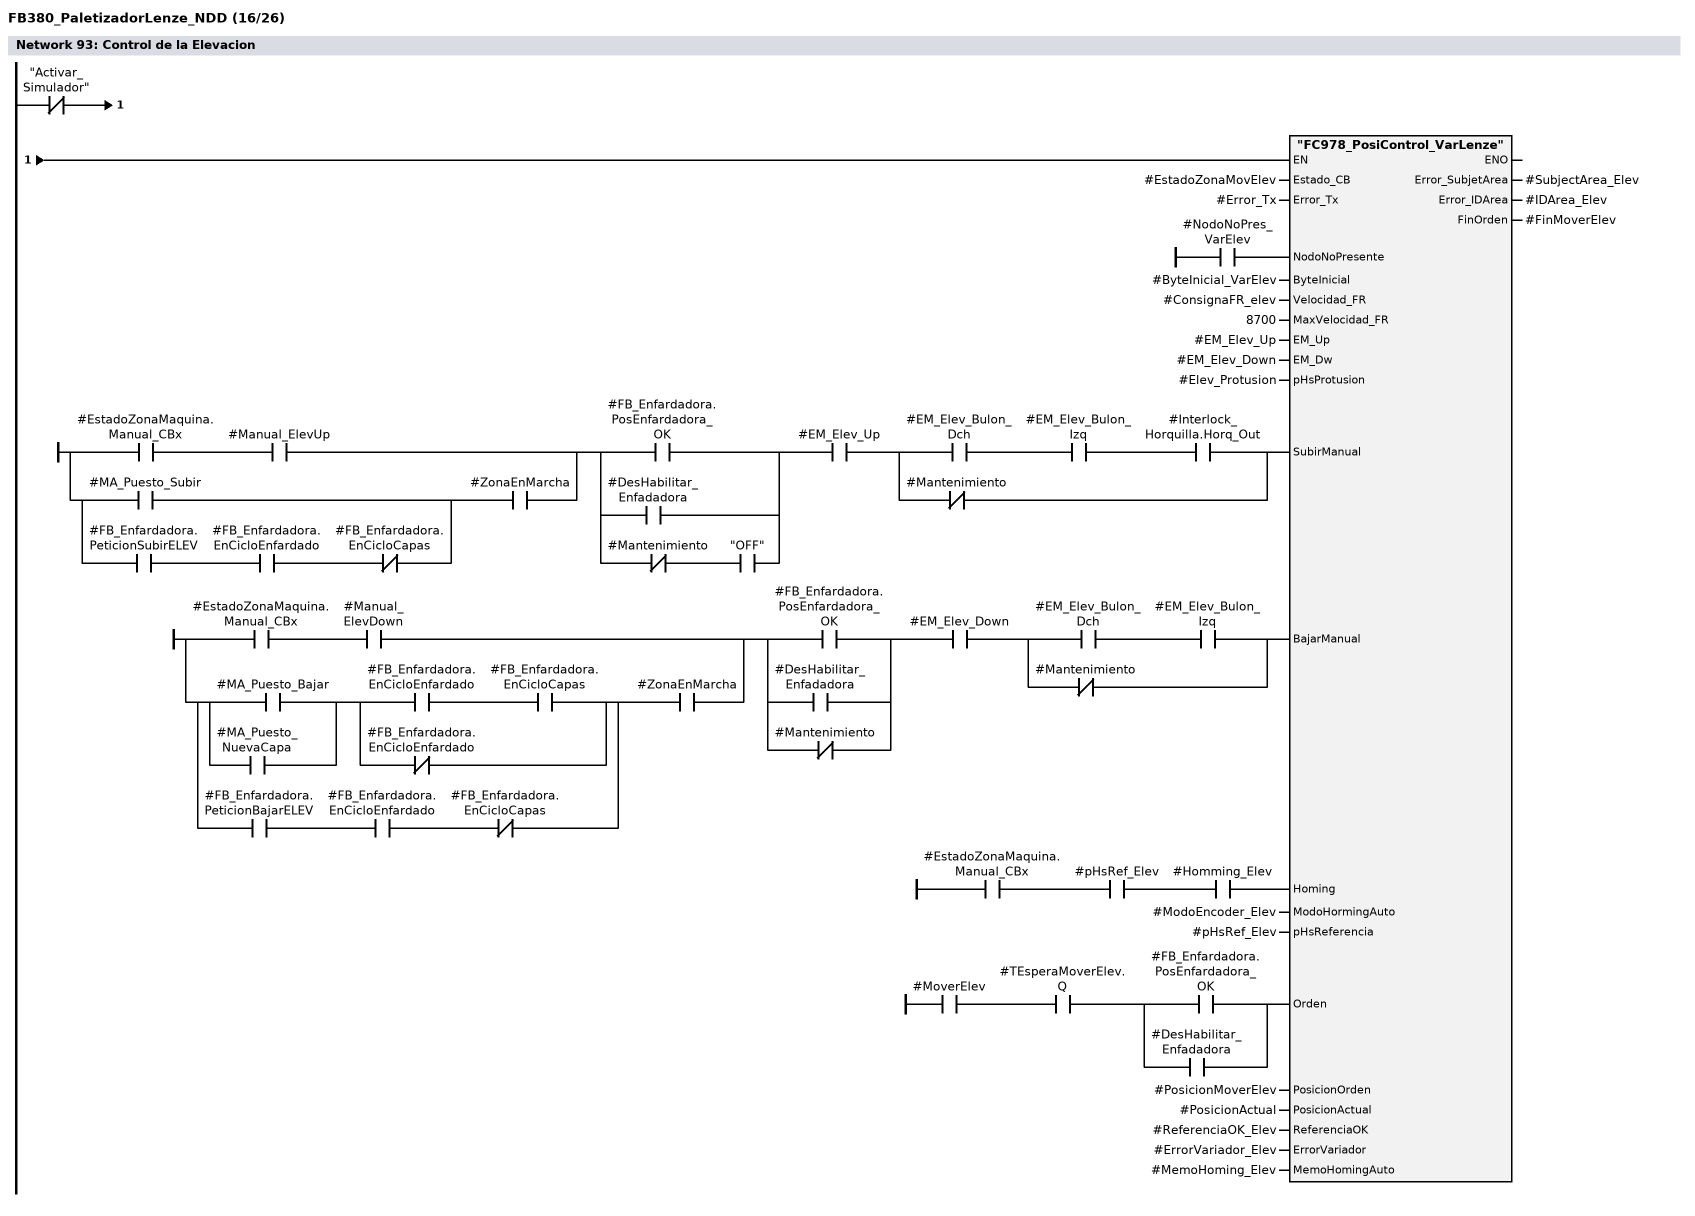
   RUNG wire#powerrail
      I_Contact( "Activar_Simulador" )
      "FC978_PosiControl_VarLenze"(NodoNoPresente := wire#w1, SubirManual := wire#w6, BajarManual := wire#w12, Homing := wire#w13, Orden := wire#w15, Estado_CB := #EstadoZonaMovElev, Error_Tx := #Error_Tx, ByteInicial := #ByteInicial_VarElev, Velocidad_FR := #ConsignaFR_elev, MaxVelocidad_FR := 8700, EM_Up := #EM_Elev_Up, EM_Dw := #EM_Elev_Down, pHsProtusion := #Elev_Protusion, ModoHormingAuto := #ModoEncoder_Elev, pHsReferencia := #pHsRef_Elev, PosicionOrden := #PosicionMoverElev, PosicionActual := #PosicionActual, ReferenciaOK := #ReferenciaOK_Elev, ErrorVariador := #ErrorVariador_Elev, MemoHomingAuto := #MemoHoming_Elev, Error_SubjetArea => #SubjectArea_Elev, Error_IDArea => #IDArea_Elev, FinOrden => #FinMoverElev)
   END_RUNG
   RUNG wire#powerrail
      Contact( #NodoNoPres_VarElev )
   END_RUNG wire#w1
   RUNG wire#powerrail
      Contact( #EstadoZonaMaquina.Manual_CBx )
      Contact( #Manual_ElevUp )
      wire#w2
      Contact( #FB_Enfardadora.PosEnfardadora_OK )
      wire#w4
      Contact( #EM_Elev_Up )
      wire#w5
      Contact( #EM_Elev_Bulon_Dch )
      Contact( #EM_Elev_Bulon_Izq )
      Contact( #Interlock_Horquilla.Horq_Out )
   END_RUNG wire#w6
   RUNG wire#powerrail
      Contact( #MA_Puesto_Subir )
      wire#w3
      Contact( #ZonaEnMarcha )
   END_RUNG wire#w2
   RUNG wire#powerrail
      Contact( #FB_Enfardadora.PeticionSubirELEV )
      Contact( #FB_Enfardadora.EnCicloEnfardado )
      I_Contact( #FB_Enfardadora.EnCicloCapas )
   END_RUNG wire#w3
   RUNG wire#w2
      Contact( #DesHabilitar_Enfadadora )
   END_RUNG wire#w4
   RUNG wire#w2
      I_Contact( #Mantenimiento )
      Contact( "OFF" )
   END_RUNG wire#w4
   RUNG wire#w5
      I_Contact( #Mantenimiento )
   END_RUNG wire#w6
   RUNG wire#powerrail
      Contact( #EstadoZonaMaquina.Manual_CBx )
      Contact( #Manual_ElevDown )
      wire#w7
      Contact( #FB_Enfardadora.PosEnfardadora_OK )
      wire#w10
      Contact( #EM_Elev_Down )
      wire#w11
      Contact( #EM_Elev_Bulon_Dch )
      Contact( #EM_Elev_Bulon_Izq )
   END_RUNG wire#w12
   RUNG wire#powerrail
      Contact( #MA_Puesto_Bajar )
      wire#w8
      Contact( #FB_Enfardadora.EnCicloEnfardado )
      Contact( #FB_Enfardadora.EnCicloCapas )
      wire#w9
      Contact( #ZonaEnMarcha )
   END_RUNG wire#w7
   RUNG wire#powerrail
      Contact( #MA_Puesto_NuevaCapa )
   END_RUNG wire#w8
   RUNG wire#w8
      I_Contact( #FB_Enfardadora.EnCicloEnfardado )
   END_RUNG wire#w9
   RUNG wire#powerrail
      Contact( #FB_Enfardadora.PeticionBajarELEV )
      Contact( #FB_Enfardadora.EnCicloEnfardado )
      I_Contact( #FB_Enfardadora.EnCicloCapas )
   END_RUNG wire#w9
   RUNG wire#w7
      Contact( #DesHabilitar_Enfadadora )
   END_RUNG wire#w10
   RUNG wire#w7
      I_Contact( #Mantenimiento )
   END_RUNG wire#w10
   RUNG wire#w11
      I_Contact( #Mantenimiento )
   END_RUNG wire#w12
   RUNG wire#powerrail
      Contact( #EstadoZonaMaquina.Manual_CBx )
      Contact( #pHsRef_Elev )
      Contact( #Homming_Elev )
   END_RUNG wire#w13
   RUNG wire#powerrail
      Contact( #MoverElev )
      Contact( #TEsperaMoverElev.Q )
      wire#w14
      Contact( #FB_Enfardadora.PosEnfardadora_OK )
   END_RUNG wire#w15
   RUNG wire#w14
      Contact( #DesHabilitar_Enfadadora )
   END_RUNG wire#w15
   // the same network as SCL:
   IF NOT "Activar_Simulador" THEN
       "FC978_PosiControl_VarLenze"(Estado_CB := #EstadoZonaMovElev,
                               Error_Tx := #Error_Tx,
                               NodoNoPresente := #NodoNoPres_VarElev,
                               ByteInicial := #ByteInicial_VarElev,
                               Velocidad_FR := #ConsignaFR_elev,
                               MaxVelocidad_FR := 8700,
                               EM_Up := #EM_Elev_Up,
                               EM_Dw := #EM_Elev_Down,
                               pHsProtusion := #Elev_Protusion,
                               SubirManual := ((#EstadoZonaMaquina.Manual_CBx AND #Manual_ElevUp) OR ((#MA_Puesto_Subir OR (#FB_Enfardadora.PeticionSubirELEV AND #FB_Enfardadora.EnCicloEnfardado AND NOT #FB_Enfardadora.EnCicloCapas)) AND #ZonaEnMarcha)) AND (#FB_Enfardadora.PosEnfardadora_OK OR #DesHabilitar_Enfadadora OR (NOT #Mantenimiento AND "OFF")) AND #EM_Elev_Up AND ((#EM_Elev_Bulon_Dch AND #EM_Elev_Bulon_Izq AND #Interlock_Horquilla.Horq_Out) OR NOT #Mantenimiento),
                               BajarManual := ((#EstadoZonaMaquina.Manual_CBx AND #Manual_ElevDown) OR ((((#MA_Puesto_Bajar OR #MA_Puesto_NuevaCapa) AND ((#FB_Enfardadora.EnCicloEnfardado AND #FB_Enfardadora.EnCicloCapas) OR NOT #FB_Enfardadora.EnCicloEnfardado)) OR (#FB_Enfardadora.PeticionBajarELEV AND #FB_Enfardadora.EnCicloEnfardado AND NOT #FB_Enfardadora.EnCicloCapas)) AND #ZonaEnMarcha)) AND (#FB_Enfardadora.PosEnfardadora_OK OR #DesHabilitar_Enfadadora OR NOT #Mantenimiento) AND #EM_Elev_Down AND ((#EM_Elev_Bulon_Dch AND #EM_Elev_Bulon_Izq) OR NOT #Mantenimiento),
                               Homing := #EstadoZonaMaquina.Manual_CBx AND #pHsRef_Elev AND #Homming_Elev,
                               ModoHormingAuto := #ModoEncoder_Elev,
                               pHsReferencia := #pHsRef_Elev,
                               Orden := #MoverElev AND #TEsperaMoverElev.Q AND (#FB_Enfardadora.PosEnfardadora_OK OR #DesHabilitar_Enfadadora),
                               PosicionOrden := #PosicionMoverElev,
                               PosicionActual := #PosicionActual,
                               ReferenciaOK := #ReferenciaOK_Elev,
                               ErrorVariador := #ErrorVariador_Elev,
                               MemoHomingAuto := #MemoHoming_Elev,
                               Error_SubjetArea => #SubjectArea_Elev,
                               Error_IDArea => #IDArea_Elev,
                               FinOrden => #FinMoverElev);
   END_IF;
END_REGION

REGION Network 94: Control de la Enfardadora
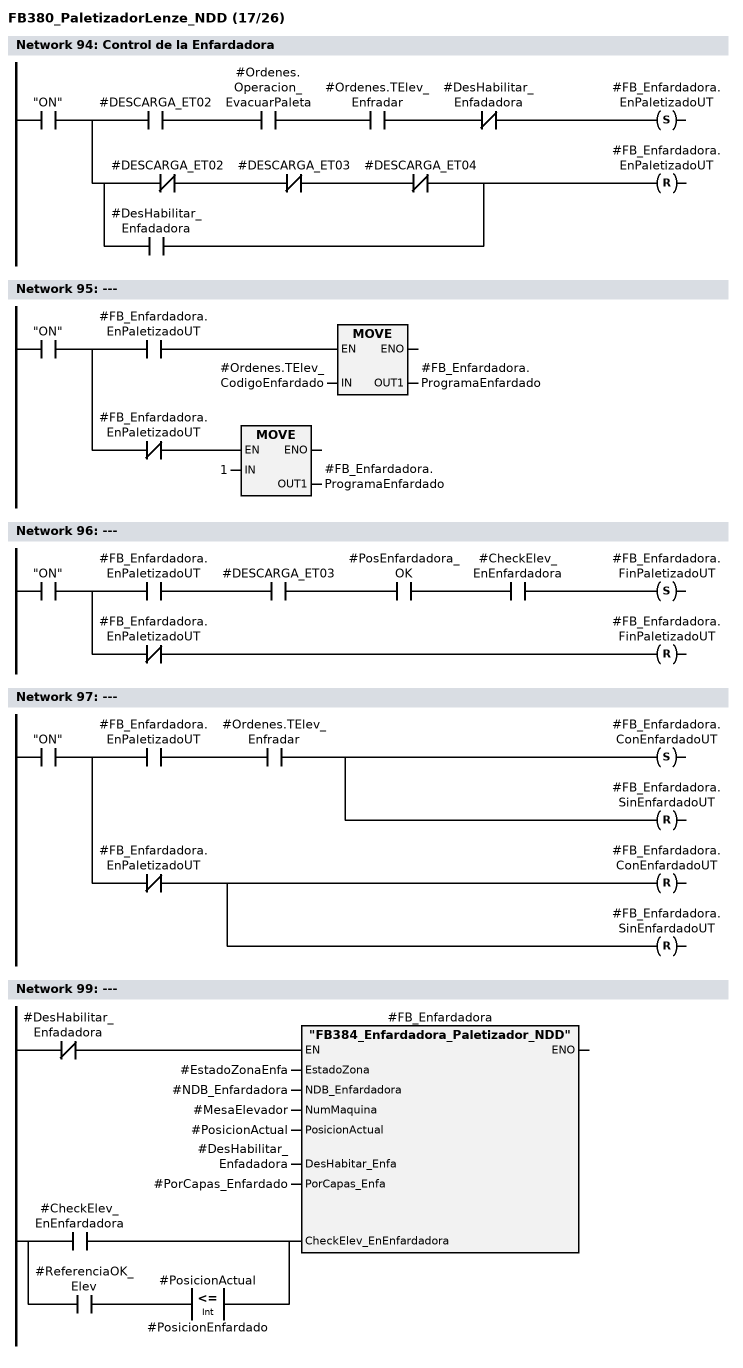
   RUNG wire#powerrail
      Contact( "ON" )
      wire#w1
      Contact( #DESCARGA_ET02 )
      Contact( #Ordenes.Operacion_EvacuarPaleta )
      Contact( #Ordenes.TElev_Enfradar )
      I_Contact( #DesHabilitar_Enfadadora )
      S_Coil( #FB_Enfardadora.EnPaletizadoUT )
   END_RUNG
   RUNG wire#w1
      I_Contact( #DESCARGA_ET02 )
      I_Contact( #DESCARGA_ET03 )
      I_Contact( #DESCARGA_ET04 )
      wire#w2
      R_Coil( #FB_Enfardadora.EnPaletizadoUT )
   END_RUNG
   RUNG wire#w1
      Contact( #DesHabilitar_Enfadadora )
   END_RUNG wire#w2
   // the same network as SCL:
   IF "ON" AND #DESCARGA_ET02 AND #Ordenes.Operacion_EvacuarPaleta AND #Ordenes.TElev_Enfradar AND NOT #DesHabilitar_Enfadadora THEN
       #FB_Enfardadora.EnPaletizadoUT := TRUE;
   END_IF;
   IF "ON" AND ((NOT #DESCARGA_ET02 AND NOT #DESCARGA_ET03 AND NOT #DESCARGA_ET04) OR #DesHabilitar_Enfadadora) THEN
       #FB_Enfardadora.EnPaletizadoUT := FALSE;
   END_IF;
END_REGION

REGION Network 95: ---
   RUNG wire#powerrail
      Contact( "ON" )
      wire#w1
      Contact( #FB_Enfardadora.EnPaletizadoUT )
      { S7_GenerateENO := "TRUE" } Move(in := #Ordenes.TElev_CodigoEnfardado, out1 => #FB_Enfardadora.ProgramaEnfardado)
   END_RUNG
   RUNG wire#w1
      I_Contact( #FB_Enfardadora.EnPaletizadoUT )
      { S7_GenerateENO := "TRUE" } Move(in := 1, out1 => #FB_Enfardadora.ProgramaEnfardado)
   END_RUNG
   // the same network as SCL:
   IF "ON" AND #FB_Enfardadora.EnPaletizadoUT THEN
       #FB_Enfardadora.ProgramaEnfardado := #Ordenes.TElev_CodigoEnfardado;
   END_IF;
   IF "ON" AND NOT #FB_Enfardadora.EnPaletizadoUT THEN #FB_Enfardadora.ProgramaEnfardado := 1; END_IF;
END_REGION

REGION Network 96: ---
   RUNG wire#powerrail
      Contact( "ON" )
      wire#w1
      Contact( #FB_Enfardadora.EnPaletizadoUT )
      Contact( #DESCARGA_ET03 )
      Contact( #PosEnfardadora_OK )
      Contact( #CheckElev_EnEnfardadora )
      S_Coil( #FB_Enfardadora.FinPaletizadoUT )
   END_RUNG
   RUNG wire#w1
      I_Contact( #FB_Enfardadora.EnPaletizadoUT )
      R_Coil( #FB_Enfardadora.FinPaletizadoUT )
   END_RUNG
   // the same network as SCL:
   IF "ON" AND #FB_Enfardadora.EnPaletizadoUT AND #DESCARGA_ET03 AND #PosEnfardadora_OK AND #CheckElev_EnEnfardadora THEN
       #FB_Enfardadora.FinPaletizadoUT := TRUE;
   END_IF;
   IF "ON" AND NOT #FB_Enfardadora.EnPaletizadoUT THEN #FB_Enfardadora.FinPaletizadoUT := FALSE; END_IF;
END_REGION

